DATA_BLOCK "IdentRfHmi"   // DB213
// stored: MemoryReserve 100
   VAR
      unitIdentRf : Array[0.."NO_OF_UNITS"] of "typeEMIdentRf";
   END_VAR
BEGIN
   unitIdentRf[0].identRfEM[0..7].selectedUnit := 0;
   unitIdentRf[0].identRfEM[0..7].selectedEM := 0;
   unitIdentRf[0].identRfEM[0..7].rfReaderId := 0;
   unitIdentRf[0].identRfEM[0..7].numberOfRf := 0;
   unitIdentRf[0].identRfEM[0].rfReader[0..1].deviceName := WSTRING#'';
   unitIdentRf[0].identRfEM[1].rfReader[0..1].deviceName := WSTRING#'';
   unitIdentRf[0].identRfEM[2].rfReader[0..1].deviceName := WSTRING#'';
   unitIdentRf[0].identRfEM[3].rfReader[0..1].deviceName := WSTRING#'';
   unitIdentRf[0].identRfEM[4].rfReader[0..1].deviceName := WSTRING#'';
   unitIdentRf[0].identRfEM[5].rfReader[0..1].deviceName := WSTRING#'';
   unitIdentRf[0].identRfEM[6].rfReader[0..1].deviceName := WSTRING#'';
   unitIdentRf[0].identRfEM[7].rfReader[0..1].deviceName := WSTRING#'';
   unitIdentRf[0].identRfEM[0].rfReader[0..1].deviceType := WSTRING#'';
   unitIdentRf[0].identRfEM[1].rfReader[0..1].deviceType := WSTRING#'';
   unitIdentRf[0].identRfEM[2].rfReader[0..1].deviceType := WSTRING#'';
   unitIdentRf[0].identRfEM[3].rfReader[0..1].deviceType := WSTRING#'';
   unitIdentRf[0].identRfEM[4].rfReader[0..1].deviceType := WSTRING#'';
   unitIdentRf[0].identRfEM[5].rfReader[0..1].deviceType := WSTRING#'';
   unitIdentRf[0].identRfEM[6].rfReader[0..1].deviceType := WSTRING#'';
   unitIdentRf[0].identRfEM[7].rfReader[0..1].deviceType := WSTRING#'';
   unitIdentRf[0].identRfEM[0].rfReader[0..1].deviceId := 0;
   unitIdentRf[0].identRfEM[1].rfReader[0..1].deviceId := 0;
   unitIdentRf[0].identRfEM[2].rfReader[0..1].deviceId := 0;
   unitIdentRf[0].identRfEM[3].rfReader[0..1].deviceId := 0;
   unitIdentRf[0].identRfEM[4].rfReader[0..1].deviceId := 0;
   unitIdentRf[0].identRfEM[5].rfReader[0..1].deviceId := 0;
   unitIdentRf[0].identRfEM[6].rfReader[0..1].deviceId := 0;
   unitIdentRf[0].identRfEM[7].rfReader[0..1].deviceId := 0;
   unitIdentRf[0].identRfEM[0].rfReader[0..1].tagType := WSTRING#'';
   unitIdentRf[0].identRfEM[1].rfReader[0..1].tagType := WSTRING#'';
   unitIdentRf[0].identRfEM[2].rfReader[0..1].tagType := WSTRING#'';
   unitIdentRf[0].identRfEM[3].rfReader[0..1].tagType := WSTRING#'';
   unitIdentRf[0].identRfEM[4].rfReader[0..1].tagType := WSTRING#'';
   unitIdentRf[0].identRfEM[5].rfReader[0..1].tagType := WSTRING#'';
   unitIdentRf[0].identRfEM[6].rfReader[0..1].tagType := WSTRING#'';
   unitIdentRf[0].identRfEM[7].rfReader[0..1].tagType := WSTRING#'';
   unitIdentRf[0].identRfEM[0].rfReader[0..1].cameraMode := WSTRING#'';
   unitIdentRf[0].identRfEM[1].rfReader[0..1].cameraMode := WSTRING#'';
   unitIdentRf[0].identRfEM[2].rfReader[0..1].cameraMode := WSTRING#'';
   unitIdentRf[0].identRfEM[3].rfReader[0..1].cameraMode := WSTRING#'';
   unitIdentRf[0].identRfEM[4].rfReader[0..1].cameraMode := WSTRING#'';
   unitIdentRf[0].identRfEM[5].rfReader[0..1].cameraMode := WSTRING#'';
   unitIdentRf[0].identRfEM[6].rfReader[0..1].cameraMode := WSTRING#'';
   unitIdentRf[0].identRfEM[7].rfReader[0..1].cameraMode := WSTRING#'';
   unitIdentRf[0].identRfEM[0].rfReader[0..1].resultState := WSTRING#'';
   unitIdentRf[0].identRfEM[1].rfReader[0..1].resultState := WSTRING#'';
   unitIdentRf[0].identRfEM[2].rfReader[0..1].resultState := WSTRING#'';
   unitIdentRf[0].identRfEM[3].rfReader[0..1].resultState := WSTRING#'';
   unitIdentRf[0].identRfEM[4].rfReader[0..1].resultState := WSTRING#'';
   unitIdentRf[0].identRfEM[5].rfReader[0..1].resultState := WSTRING#'';
   unitIdentRf[0].identRfEM[6].rfReader[0..1].resultState := WSTRING#'';
   unitIdentRf[0].identRfEM[7].rfReader[0..1].resultState := WSTRING#'';
   unitIdentRf[0].identRfEM[0].rfReader[0..1].progNo := 0;
   unitIdentRf[0].identRfEM[1].rfReader[0..1].progNo := 0;
   unitIdentRf[0].identRfEM[2].rfReader[0..1].progNo := 0;
   unitIdentRf[0].identRfEM[3].rfReader[0..1].progNo := 0;
   unitIdentRf[0].identRfEM[4].rfReader[0..1].progNo := 0;
   unitIdentRf[0].identRfEM[5].rfReader[0..1].progNo := 0;
   unitIdentRf[0].identRfEM[6].rfReader[0..1].progNo := 0;
   unitIdentRf[0].identRfEM[7].rfReader[0..1].progNo := 0;
   unitIdentRf[0].identRfEM[0].rfReader[0..1].progNumberWrite := 0;
   unitIdentRf[0].identRfEM[1].rfReader[0..1].progNumberWrite := 0;
   unitIdentRf[0].identRfEM[2].rfReader[0..1].progNumberWrite := 0;
   unitIdentRf[0].identRfEM[3].rfReader[0..1].progNumberWrite := 0;
   unitIdentRf[0].identRfEM[4].rfReader[0..1].progNumberWrite := 0;
   unitIdentRf[0].identRfEM[5].rfReader[0..1].progNumberWrite := 0;
   unitIdentRf[0].identRfEM[6].rfReader[0..1].progNumberWrite := 0;
   unitIdentRf[0].identRfEM[7].rfReader[0..1].progNumberWrite := 0;
   unitIdentRf[0].identRfEM[0].rfReader[0..1].pushbutton := 16#0000;
   unitIdentRf[0].identRfEM[1].rfReader[0..1].pushbutton := 16#0000;
   unitIdentRf[0].identRfEM[2].rfReader[0..1].pushbutton := 16#0000;
   unitIdentRf[0].identRfEM[3].rfReader[0..1].pushbutton := 16#0000;
   unitIdentRf[0].identRfEM[4].rfReader[0..1].pushbutton := 16#0000;
   unitIdentRf[0].identRfEM[5].rfReader[0..1].pushbutton := 16#0000;
   unitIdentRf[0].identRfEM[6].rfReader[0..1].pushbutton := 16#0000;
   unitIdentRf[0].identRfEM[7].rfReader[0..1].pushbutton := 16#0000;
   unitIdentRf[0].identRfEM[0].rfReader[0..1].enablePushbutton := 16#0000;
   unitIdentRf[0].identRfEM[1].rfReader[0..1].enablePushbutton := 16#0000;
   unitIdentRf[0].identRfEM[2].rfReader[0..1].enablePushbutton := 16#0000;
   unitIdentRf[0].identRfEM[3].rfReader[0..1].enablePushbutton := 16#0000;
   unitIdentRf[0].identRfEM[4].rfReader[0..1].enablePushbutton := 16#0000;
   unitIdentRf[0].identRfEM[5].rfReader[0..1].enablePushbutton := 16#0000;
   unitIdentRf[0].identRfEM[6].rfReader[0..1].enablePushbutton := 16#0000;
   unitIdentRf[0].identRfEM[7].rfReader[0..1].enablePushbutton := 16#0000;
   unitIdentRf[0].identRfEM[0].rfReader[0..1].status := 16#0000;
   unitIdentRf[0].identRfEM[1].rfReader[0..1].status := 16#0000;
   unitIdentRf[0].identRfEM[2].rfReader[0..1].status := 16#0000;
   unitIdentRf[0].identRfEM[3].rfReader[0..1].status := 16#0000;
   unitIdentRf[0].identRfEM[4].rfReader[0..1].status := 16#0000;
   unitIdentRf[0].identRfEM[5].rfReader[0..1].status := 16#0000;
   unitIdentRf[0].identRfEM[6].rfReader[0..1].status := 16#0000;
   unitIdentRf[0].identRfEM[7].rfReader[0..1].status := 16#0000;
   unitIdentRf[0].identRfEM[0].rfReader[0..1].alarmCategorie := 0;
   unitIdentRf[0].identRfEM[1].rfReader[0..1].alarmCategorie := 0;
   unitIdentRf[0].identRfEM[2].rfReader[0..1].alarmCategorie := 0;
   unitIdentRf[0].identRfEM[3].rfReader[0..1].alarmCategorie := 0;
   unitIdentRf[0].identRfEM[4].rfReader[0..1].alarmCategorie := 0;
   unitIdentRf[0].identRfEM[5].rfReader[0..1].alarmCategorie := 0;
   unitIdentRf[0].identRfEM[6].rfReader[0..1].alarmCategorie := 0;
   unitIdentRf[0].identRfEM[7].rfReader[0..1].alarmCategorie := 0;
   unitIdentRf[0].identRfEM[0].rfReader[0..1].alarmNo := 0;
   unitIdentRf[0].identRfEM[1].rfReader[0..1].alarmNo := 0;
   unitIdentRf[0].identRfEM[2].rfReader[0..1].alarmNo := 0;
   unitIdentRf[0].identRfEM[3].rfReader[0..1].alarmNo := 0;
   unitIdentRf[0].identRfEM[4].rfReader[0..1].alarmNo := 0;
   unitIdentRf[0].identRfEM[5].rfReader[0..1].alarmNo := 0;
   unitIdentRf[0].identRfEM[6].rfReader[0..1].alarmNo := 0;
   unitIdentRf[0].identRfEM[7].rfReader[0..1].alarmNo := 0;
   unitIdentRf[0].identRfEM[0].rfReader[0..1].alarmCode := 16#0000_0000;
   unitIdentRf[0].identRfEM[1].rfReader[0..1].alarmCode := 16#0000_0000;
   unitIdentRf[0].identRfEM[2].rfReader[0..1].alarmCode := 16#0000_0000;
   unitIdentRf[0].identRfEM[3].rfReader[0..1].alarmCode := 16#0000_0000;
   unitIdentRf[0].identRfEM[4].rfReader[0..1].alarmCode := 16#0000_0000;
   unitIdentRf[0].identRfEM[5].rfReader[0..1].alarmCode := 16#0000_0000;
   unitIdentRf[0].identRfEM[6].rfReader[0..1].alarmCode := 16#0000_0000;
   unitIdentRf[0].identRfEM[7].rfReader[0..1].alarmCode := 16#0000_0000;
   unitIdentRf[0].identRfEM[0].rfReader[0..1].resultColor := 0;
   unitIdentRf[0].identRfEM[1].rfReader[0..1].resultColor := 0;
   unitIdentRf[0].identRfEM[2].rfReader[0..1].resultColor := 0;
   unitIdentRf[0].identRfEM[3].rfReader[0..1].resultColor := 0;
   unitIdentRf[0].identRfEM[4].rfReader[0..1].resultColor := 0;
   unitIdentRf[0].identRfEM[5].rfReader[0..1].resultColor := 0;
   unitIdentRf[0].identRfEM[6].rfReader[0..1].resultColor := 0;
   unitIdentRf[0].identRfEM[7].rfReader[0..1].resultColor := 0;
   unitIdentRf[0].identRfEM[0].rfReader[0..1].statusColorCode := 0;
   unitIdentRf[0].identRfEM[1].rfReader[0..1].statusColorCode := 0;
   unitIdentRf[0].identRfEM[2].rfReader[0..1].statusColorCode := 0;
   unitIdentRf[0].identRfEM[3].rfReader[0..1].statusColorCode := 0;
   unitIdentRf[0].identRfEM[4].rfReader[0..1].statusColorCode := 0;
   unitIdentRf[0].identRfEM[5].rfReader[0..1].statusColorCode := 0;
   unitIdentRf[0].identRfEM[6].rfReader[0..1].statusColorCode := 0;
   unitIdentRf[0].identRfEM[7].rfReader[0..1].statusColorCode := 0;
   unitIdentRf[0].identRfEM[0].rfReader[0..1].datRead1 := '';
   unitIdentRf[0].identRfEM[1].rfReader[0..1].datRead1 := '';
   unitIdentRf[0].identRfEM[2].rfReader[0..1].datRead1 := '';
   unitIdentRf[0].identRfEM[3].rfReader[0..1].datRead1 := '';
   unitIdentRf[0].identRfEM[4].rfReader[0..1].datRead1 := '';
   unitIdentRf[0].identRfEM[5].rfReader[0..1].datRead1 := '';
   unitIdentRf[0].identRfEM[6].rfReader[0..1].datRead1 := '';
   unitIdentRf[0].identRfEM[7].rfReader[0..1].datRead1 := '';
   unitIdentRf[0].identRfEM[0].rfReader[0..1].datRead2 := '';
   unitIdentRf[0].identRfEM[1].rfReader[0..1].datRead2 := '';
   unitIdentRf[0].identRfEM[2].rfReader[0..1].datRead2 := '';
   unitIdentRf[0].identRfEM[3].rfReader[0..1].datRead2 := '';
   unitIdentRf[0].identRfEM[4].rfReader[0..1].datRead2 := '';
   unitIdentRf[0].identRfEM[5].rfReader[0..1].datRead2 := '';
   unitIdentRf[0].identRfEM[6].rfReader[0..1].datRead2 := '';
   unitIdentRf[0].identRfEM[7].rfReader[0..1].datRead2 := '';
   unitIdentRf[0].identRfEM[0].rfReader[0..1].datRead3 := '';
   unitIdentRf[0].identRfEM[1].rfReader[0..1].datRead3 := '';
   unitIdentRf[0].identRfEM[2].rfReader[0..1].datRead3 := '';
   unitIdentRf[0].identRfEM[3].rfReader[0..1].datRead3 := '';
   unitIdentRf[0].identRfEM[4].rfReader[0..1].datRead3 := '';
   unitIdentRf[0].identRfEM[5].rfReader[0..1].datRead3 := '';
   unitIdentRf[0].identRfEM[6].rfReader[0..1].datRead3 := '';
   unitIdentRf[0].identRfEM[7].rfReader[0..1].datRead3 := '';
   unitIdentRf[0].identRfEM[0].rfReader[0..1].datRead4 := '';
   unitIdentRf[0].identRfEM[1].rfReader[0..1].datRead4 := '';
   unitIdentRf[0].identRfEM[2].rfReader[0..1].datRead4 := '';
   unitIdentRf[0].identRfEM[3].rfReader[0..1].datRead4 := '';
   unitIdentRf[0].identRfEM[4].rfReader[0..1].datRead4 := '';
   unitIdentRf[0].identRfEM[5].rfReader[0..1].datRead4 := '';
   unitIdentRf[0].identRfEM[6].rfReader[0..1].datRead4 := '';
   unitIdentRf[0].identRfEM[7].rfReader[0..1].datRead4 := '';
   unitIdentRf[0].identRfEM[0].rfReader[0..1].datWrite1 := '';
   unitIdentRf[0].identRfEM[1].rfReader[0..1].datWrite1 := '';
   unitIdentRf[0].identRfEM[2].rfReader[0..1].datWrite1 := '';
   unitIdentRf[0].identRfEM[3].rfReader[0..1].datWrite1 := '';
   unitIdentRf[0].identRfEM[4].rfReader[0..1].datWrite1 := '';
   unitIdentRf[0].identRfEM[5].rfReader[0..1].datWrite1 := '';
   unitIdentRf[0].identRfEM[6].rfReader[0..1].datWrite1 := '';
   unitIdentRf[0].identRfEM[7].rfReader[0..1].datWrite1 := '';
   unitIdentRf[0].identRfEM[0].rfReader[0..1].datWrite2 := '';
   unitIdentRf[0].identRfEM[1].rfReader[0..1].datWrite2 := '';
   unitIdentRf[0].identRfEM[2].rfReader[0..1].datWrite2 := '';
   unitIdentRf[0].identRfEM[3].rfReader[0..1].datWrite2 := '';
   unitIdentRf[0].identRfEM[4].rfReader[0..1].datWrite2 := '';
   unitIdentRf[0].identRfEM[5].rfReader[0..1].datWrite2 := '';
   unitIdentRf[0].identRfEM[6].rfReader[0..1].datWrite2 := '';
   unitIdentRf[0].identRfEM[7].rfReader[0..1].datWrite2 := '';
   unitIdentRf[0].identRfEM[0].rfReader[0..1].datWrite3 := '';
   unitIdentRf[0].identRfEM[1].rfReader[0..1].datWrite3 := '';
   unitIdentRf[0].identRfEM[2].rfReader[0..1].datWrite3 := '';
   unitIdentRf[0].identRfEM[3].rfReader[0..1].datWrite3 := '';
   unitIdentRf[0].identRfEM[4].rfReader[0..1].datWrite3 := '';
   unitIdentRf[0].identRfEM[5].rfReader[0..1].datWrite3 := '';
   unitIdentRf[0].identRfEM[6].rfReader[0..1].datWrite3 := '';
   unitIdentRf[0].identRfEM[7].rfReader[0..1].datWrite3 := '';
   unitIdentRf[0].identRfEM[0].rfReader[0..1].datWrite4 := '';
   unitIdentRf[0].identRfEM[1].rfReader[0..1].datWrite4 := '';
   unitIdentRf[0].identRfEM[2].rfReader[0..1].datWrite4 := '';
   unitIdentRf[0].identRfEM[3].rfReader[0..1].datWrite4 := '';
   unitIdentRf[0].identRfEM[4].rfReader[0..1].datWrite4 := '';
   unitIdentRf[0].identRfEM[5].rfReader[0..1].datWrite4 := '';
   unitIdentRf[0].identRfEM[6].rfReader[0..1].datWrite4 := '';
   unitIdentRf[0].identRfEM[7].rfReader[0..1].datWrite4 := '';
END_DATA_BLOCK

DATA_BLOCK "IdentMvHmi"   // DB214
// stored: MemoryReserve 100
   VAR
      unitIdentMv : Array[0.."NO_OF_UNITS"] of "typeEMIdentMv";
   END_VAR
BEGIN
   unitIdentMv[0].identMvEM[0..7].selectedUnit := 0;
   unitIdentMv[0].identMvEM[0..7].selectedEM := 0;
   unitIdentMv[0].identMvEM[0..7].mvReaderId := 0;
   unitIdentMv[0].identMvEM[0..7].numberOfMv := 0;
   unitIdentMv[0].identMvEM[0].mvReader[0..1].deviceName := WSTRING#'';
   unitIdentMv[0].identMvEM[1].mvReader[0..1].deviceName := WSTRING#'';
   unitIdentMv[0].identMvEM[2].mvReader[0..1].deviceName := WSTRING#'';
   unitIdentMv[0].identMvEM[3].mvReader[0..1].deviceName := WSTRING#'';
   unitIdentMv[0].identMvEM[4].mvReader[0..1].deviceName := WSTRING#'';
   unitIdentMv[0].identMvEM[5].mvReader[0..1].deviceName := WSTRING#'';
   unitIdentMv[0].identMvEM[6].mvReader[0..1].deviceName := WSTRING#'';
   unitIdentMv[0].identMvEM[7].mvReader[0..1].deviceName := WSTRING#'';
   unitIdentMv[0].identMvEM[0].mvReader[0..1].deviceType := WSTRING#'';
   unitIdentMv[0].identMvEM[1].mvReader[0..1].deviceType := WSTRING#'';
   unitIdentMv[0].identMvEM[2].mvReader[0..1].deviceType := WSTRING#'';
   unitIdentMv[0].identMvEM[3].mvReader[0..1].deviceType := WSTRING#'';
   unitIdentMv[0].identMvEM[4].mvReader[0..1].deviceType := WSTRING#'';
   unitIdentMv[0].identMvEM[5].mvReader[0..1].deviceType := WSTRING#'';
   unitIdentMv[0].identMvEM[6].mvReader[0..1].deviceType := WSTRING#'';
   unitIdentMv[0].identMvEM[7].mvReader[0..1].deviceType := WSTRING#'';
   unitIdentMv[0].identMvEM[0].mvReader[0..1].deviceId := 0;
   unitIdentMv[0].identMvEM[1].mvReader[0..1].deviceId := 0;
   unitIdentMv[0].identMvEM[2].mvReader[0..1].deviceId := 0;
   unitIdentMv[0].identMvEM[3].mvReader[0..1].deviceId := 0;
   unitIdentMv[0].identMvEM[4].mvReader[0..1].deviceId := 0;
   unitIdentMv[0].identMvEM[5].mvReader[0..1].deviceId := 0;
   unitIdentMv[0].identMvEM[6].mvReader[0..1].deviceId := 0;
   unitIdentMv[0].identMvEM[7].mvReader[0..1].deviceId := 0;
   unitIdentMv[0].identMvEM[0].mvReader[0..1].tagType := WSTRING#'';
   unitIdentMv[0].identMvEM[1].mvReader[0..1].tagType := WSTRING#'';
   unitIdentMv[0].identMvEM[2].mvReader[0..1].tagType := WSTRING#'';
   unitIdentMv[0].identMvEM[3].mvReader[0..1].tagType := WSTRING#'';
   unitIdentMv[0].identMvEM[4].mvReader[0..1].tagType := WSTRING#'';
   unitIdentMv[0].identMvEM[5].mvReader[0..1].tagType := WSTRING#'';
   unitIdentMv[0].identMvEM[6].mvReader[0..1].tagType := WSTRING#'';
   unitIdentMv[0].identMvEM[7].mvReader[0..1].tagType := WSTRING#'';
   unitIdentMv[0].identMvEM[0].mvReader[0..1].cameraMode := WSTRING#'';
   unitIdentMv[0].identMvEM[1].mvReader[0..1].cameraMode := WSTRING#'';
   unitIdentMv[0].identMvEM[2].mvReader[0..1].cameraMode := WSTRING#'';
   unitIdentMv[0].identMvEM[3].mvReader[0..1].cameraMode := WSTRING#'';
   unitIdentMv[0].identMvEM[4].mvReader[0..1].cameraMode := WSTRING#'';
   unitIdentMv[0].identMvEM[5].mvReader[0..1].cameraMode := WSTRING#'';
   unitIdentMv[0].identMvEM[6].mvReader[0..1].cameraMode := WSTRING#'';
   unitIdentMv[0].identMvEM[7].mvReader[0..1].cameraMode := WSTRING#'';
   unitIdentMv[0].identMvEM[0].mvReader[0..1].resultState := WSTRING#'';
   unitIdentMv[0].identMvEM[1].mvReader[0..1].resultState := WSTRING#'';
   unitIdentMv[0].identMvEM[2].mvReader[0..1].resultState := WSTRING#'';
   unitIdentMv[0].identMvEM[3].mvReader[0..1].resultState := WSTRING#'';
   unitIdentMv[0].identMvEM[4].mvReader[0..1].resultState := WSTRING#'';
   unitIdentMv[0].identMvEM[5].mvReader[0..1].resultState := WSTRING#'';
   unitIdentMv[0].identMvEM[6].mvReader[0..1].resultState := WSTRING#'';
   unitIdentMv[0].identMvEM[7].mvReader[0..1].resultState := WSTRING#'';
   unitIdentMv[0].identMvEM[0].mvReader[0..1].progNo := 0;
   unitIdentMv[0].identMvEM[1].mvReader[0..1].progNo := 0;
   unitIdentMv[0].identMvEM[2].mvReader[0..1].progNo := 0;
   unitIdentMv[0].identMvEM[3].mvReader[0..1].progNo := 0;
   unitIdentMv[0].identMvEM[4].mvReader[0..1].progNo := 0;
   unitIdentMv[0].identMvEM[5].mvReader[0..1].progNo := 0;
   unitIdentMv[0].identMvEM[6].mvReader[0..1].progNo := 0;
   unitIdentMv[0].identMvEM[7].mvReader[0..1].progNo := 0;
   unitIdentMv[0].identMvEM[0].mvReader[0..1].progNumberWrite := 0;
   unitIdentMv[0].identMvEM[1].mvReader[0..1].progNumberWrite := 0;
   unitIdentMv[0].identMvEM[2].mvReader[0..1].progNumberWrite := 0;
   unitIdentMv[0].identMvEM[3].mvReader[0..1].progNumberWrite := 0;
   unitIdentMv[0].identMvEM[4].mvReader[0..1].progNumberWrite := 0;
   unitIdentMv[0].identMvEM[5].mvReader[0..1].progNumberWrite := 0;
   unitIdentMv[0].identMvEM[6].mvReader[0..1].progNumberWrite := 0;
   unitIdentMv[0].identMvEM[7].mvReader[0..1].progNumberWrite := 0;
   unitIdentMv[0].identMvEM[0].mvReader[0..1].pushbutton := 16#0000;
   unitIdentMv[0].identMvEM[1].mvReader[0..1].pushbutton := 16#0000;
   unitIdentMv[0].identMvEM[2].mvReader[0..1].pushbutton := 16#0000;
   unitIdentMv[0].identMvEM[3].mvReader[0..1].pushbutton := 16#0000;
   unitIdentMv[0].identMvEM[4].mvReader[0..1].pushbutton := 16#0000;
   unitIdentMv[0].identMvEM[5].mvReader[0..1].pushbutton := 16#0000;
   unitIdentMv[0].identMvEM[6].mvReader[0..1].pushbutton := 16#0000;
   unitIdentMv[0].identMvEM[7].mvReader[0..1].pushbutton := 16#0000;
   unitIdentMv[0].identMvEM[0].mvReader[0..1].enablePushbutton := 16#0000;
   unitIdentMv[0].identMvEM[1].mvReader[0..1].enablePushbutton := 16#0000;
   unitIdentMv[0].identMvEM[2].mvReader[0..1].enablePushbutton := 16#0000;
   unitIdentMv[0].identMvEM[3].mvReader[0..1].enablePushbutton := 16#0000;
   unitIdentMv[0].identMvEM[4].mvReader[0..1].enablePushbutton := 16#0000;
   unitIdentMv[0].identMvEM[5].mvReader[0..1].enablePushbutton := 16#0000;
   unitIdentMv[0].identMvEM[6].mvReader[0..1].enablePushbutton := 16#0000;
   unitIdentMv[0].identMvEM[7].mvReader[0..1].enablePushbutton := 16#0000;
   unitIdentMv[0].identMvEM[0].mvReader[0..1].status := 16#0000;
   unitIdentMv[0].identMvEM[1].mvReader[0..1].status := 16#0000;
   unitIdentMv[0].identMvEM[2].mvReader[0..1].status := 16#0000;
   unitIdentMv[0].identMvEM[3].mvReader[0..1].status := 16#0000;
   unitIdentMv[0].identMvEM[4].mvReader[0..1].status := 16#0000;
   unitIdentMv[0].identMvEM[5].mvReader[0..1].status := 16#0000;
   unitIdentMv[0].identMvEM[6].mvReader[0..1].status := 16#0000;
   unitIdentMv[0].identMvEM[7].mvReader[0..1].status := 16#0000;
   unitIdentMv[0].identMvEM[0].mvReader[0..1].alarmCategorie := 0;
   unitIdentMv[0].identMvEM[1].mvReader[0..1].alarmCategorie := 0;
   unitIdentMv[0].identMvEM[2].mvReader[0..1].alarmCategorie := 0;
   unitIdentMv[0].identMvEM[3].mvReader[0..1].alarmCategorie := 0;
   unitIdentMv[0].identMvEM[4].mvReader[0..1].alarmCategorie := 0;
   unitIdentMv[0].identMvEM[5].mvReader[0..1].alarmCategorie := 0;
   unitIdentMv[0].identMvEM[6].mvReader[0..1].alarmCategorie := 0;
   unitIdentMv[0].identMvEM[7].mvReader[0..1].alarmCategorie := 0;
   unitIdentMv[0].identMvEM[0].mvReader[0..1].alarmNo := 0;
   unitIdentMv[0].identMvEM[1].mvReader[0..1].alarmNo := 0;
   unitIdentMv[0].identMvEM[2].mvReader[0..1].alarmNo := 0;
   unitIdentMv[0].identMvEM[3].mvReader[0..1].alarmNo := 0;
   unitIdentMv[0].identMvEM[4].mvReader[0..1].alarmNo := 0;
   unitIdentMv[0].identMvEM[5].mvReader[0..1].alarmNo := 0;
   unitIdentMv[0].identMvEM[6].mvReader[0..1].alarmNo := 0;
   unitIdentMv[0].identMvEM[7].mvReader[0..1].alarmNo := 0;
   unitIdentMv[0].identMvEM[0].mvReader[0..1].alarmCode := 16#0000_0000;
   unitIdentMv[0].identMvEM[1].mvReader[0..1].alarmCode := 16#0000_0000;
   unitIdentMv[0].identMvEM[2].mvReader[0..1].alarmCode := 16#0000_0000;
   unitIdentMv[0].identMvEM[3].mvReader[0..1].alarmCode := 16#0000_0000;
   unitIdentMv[0].identMvEM[4].mvReader[0..1].alarmCode := 16#0000_0000;
   unitIdentMv[0].identMvEM[5].mvReader[0..1].alarmCode := 16#0000_0000;
   unitIdentMv[0].identMvEM[6].mvReader[0..1].alarmCode := 16#0000_0000;
   unitIdentMv[0].identMvEM[7].mvReader[0..1].alarmCode := 16#0000_0000;
   unitIdentMv[0].identMvEM[0].mvReader[0..1].resultColor := 0;
   unitIdentMv[0].identMvEM[1].mvReader[0..1].resultColor := 0;
   unitIdentMv[0].identMvEM[2].mvReader[0..1].resultColor := 0;
   unitIdentMv[0].identMvEM[3].mvReader[0..1].resultColor := 0;
   unitIdentMv[0].identMvEM[4].mvReader[0..1].resultColor := 0;
   unitIdentMv[0].identMvEM[5].mvReader[0..1].resultColor := 0;
   unitIdentMv[0].identMvEM[6].mvReader[0..1].resultColor := 0;
   unitIdentMv[0].identMvEM[7].mvReader[0..1].resultColor := 0;
   unitIdentMv[0].identMvEM[0].mvReader[0..1].statusColorCode := 0;
   unitIdentMv[0].identMvEM[1].mvReader[0..1].statusColorCode := 0;
   unitIdentMv[0].identMvEM[2].mvReader[0..1].statusColorCode := 0;
   unitIdentMv[0].identMvEM[3].mvReader[0..1].statusColorCode := 0;
   unitIdentMv[0].identMvEM[4].mvReader[0..1].statusColorCode := 0;
   unitIdentMv[0].identMvEM[5].mvReader[0..1].statusColorCode := 0;
   unitIdentMv[0].identMvEM[6].mvReader[0..1].statusColorCode := 0;
   unitIdentMv[0].identMvEM[7].mvReader[0..1].statusColorCode := 0;
   unitIdentMv[0].identMvEM[0].mvReader[0..1].datRead1 := '';
   unitIdentMv[0].identMvEM[1].mvReader[0..1].datRead1 := '';
   unitIdentMv[0].identMvEM[2].mvReader[0..1].datRead1 := '';
   unitIdentMv[0].identMvEM[3].mvReader[0..1].datRead1 := '';
   unitIdentMv[0].identMvEM[4].mvReader[0..1].datRead1 := '';
   unitIdentMv[0].identMvEM[5].mvReader[0..1].datRead1 := '';
   unitIdentMv[0].identMvEM[6].mvReader[0..1].datRead1 := '';
   unitIdentMv[0].identMvEM[7].mvReader[0..1].datRead1 := '';
   unitIdentMv[0].identMvEM[0].mvReader[0..1].datRead2 := '';
   unitIdentMv[0].identMvEM[1].mvReader[0..1].datRead2 := '';
   unitIdentMv[0].identMvEM[2].mvReader[0..1].datRead2 := '';
   unitIdentMv[0].identMvEM[3].mvReader[0..1].datRead2 := '';
   unitIdentMv[0].identMvEM[4].mvReader[0..1].datRead2 := '';
   unitIdentMv[0].identMvEM[5].mvReader[0..1].datRead2 := '';
   unitIdentMv[0].identMvEM[6].mvReader[0..1].datRead2 := '';
   unitIdentMv[0].identMvEM[7].mvReader[0..1].datRead2 := '';
   unitIdentMv[0].identMvEM[0].mvReader[0..1].datRead3 := '';
   unitIdentMv[0].identMvEM[1].mvReader[0..1].datRead3 := '';
   unitIdentMv[0].identMvEM[2].mvReader[0..1].datRead3 := '';
   unitIdentMv[0].identMvEM[3].mvReader[0..1].datRead3 := '';
   unitIdentMv[0].identMvEM[4].mvReader[0..1].datRead3 := '';
   unitIdentMv[0].identMvEM[5].mvReader[0..1].datRead3 := '';
   unitIdentMv[0].identMvEM[6].mvReader[0..1].datRead3 := '';
   unitIdentMv[0].identMvEM[7].mvReader[0..1].datRead3 := '';
   unitIdentMv[0].identMvEM[0].mvReader[0..1].datRead4 := '';
   unitIdentMv[0].identMvEM[1].mvReader[0..1].datRead4 := '';
   unitIdentMv[0].identMvEM[2].mvReader[0..1].datRead4 := '';
   unitIdentMv[0].identMvEM[3].mvReader[0..1].datRead4 := '';
   unitIdentMv[0].identMvEM[4].mvReader[0..1].datRead4 := '';
   unitIdentMv[0].identMvEM[5].mvReader[0..1].datRead4 := '';
   unitIdentMv[0].identMvEM[6].mvReader[0..1].datRead4 := '';
   unitIdentMv[0].identMvEM[7].mvReader[0..1].datRead4 := '';
   unitIdentMv[0].identMvEM[0].mvReader[0].datWrite1 := '';
   unitIdentMv[0].identMvEM[0].mvReader[1].datWrite1 := 'Siemens';
   unitIdentMv[0].identMvEM[1].mvReader[0..1].datWrite1 := '';
   unitIdentMv[0].identMvEM[2].mvReader[0..1].datWrite1 := '';
   unitIdentMv[0].identMvEM[3].mvReader[0..1].datWrite1 := '';
   unitIdentMv[0].identMvEM[4].mvReader[0..1].datWrite1 := '';
   unitIdentMv[0].identMvEM[5].mvReader[0..1].datWrite1 := '';
   unitIdentMv[0].identMvEM[6].mvReader[0..1].datWrite1 := '';
   unitIdentMv[0].identMvEM[7].mvReader[0..1].datWrite1 := '';
   unitIdentMv[0].identMvEM[0].mvReader[0..1].datWrite2 := '';
   unitIdentMv[0].identMvEM[1].mvReader[0..1].datWrite2 := '';
   unitIdentMv[0].identMvEM[2].mvReader[0..1].datWrite2 := '';
   unitIdentMv[0].identMvEM[3].mvReader[0..1].datWrite2 := '';
   unitIdentMv[0].identMvEM[4].mvReader[0..1].datWrite2 := '';
   unitIdentMv[0].identMvEM[5].mvReader[0..1].datWrite2 := '';
   unitIdentMv[0].identMvEM[6].mvReader[0..1].datWrite2 := '';
   unitIdentMv[0].identMvEM[7].mvReader[0..1].datWrite2 := '';
   unitIdentMv[0].identMvEM[0].mvReader[0..1].datWrite3 := '';
   unitIdentMv[0].identMvEM[1].mvReader[0..1].datWrite3 := '';
   unitIdentMv[0].identMvEM[2].mvReader[0..1].datWrite3 := '';
   unitIdentMv[0].identMvEM[3].mvReader[0..1].datWrite3 := '';
   unitIdentMv[0].identMvEM[4].mvReader[0..1].datWrite3 := '';
   unitIdentMv[0].identMvEM[5].mvReader[0..1].datWrite3 := '';
   unitIdentMv[0].identMvEM[6].mvReader[0..1].datWrite3 := '';
   unitIdentMv[0].identMvEM[7].mvReader[0..1].datWrite3 := '';
   unitIdentMv[0].identMvEM[0].mvReader[0..1].datWrite4 := '';
   unitIdentMv[0].identMvEM[1].mvReader[0..1].datWrite4 := '';
   unitIdentMv[0].identMvEM[2].mvReader[0..1].datWrite4 := '';
   unitIdentMv[0].identMvEM[3].mvReader[0..1].datWrite4 := '';
   unitIdentMv[0].identMvEM[4].mvReader[0..1].datWrite4 := '';
   unitIdentMv[0].identMvEM[5].mvReader[0..1].datWrite4 := '';
   unitIdentMv[0].identMvEM[6].mvReader[0..1].datWrite4 := '';
   unitIdentMv[0].identMvEM[7].mvReader[0..1].datWrite4 := '';
END_DATA_BLOCK

DATA_BLOCK "BK02"   // DB304
// stored: MemoryReserve 100
   VAR
      "X10-1.SUCTION PAD TOP DOWN" : Bool := TRUE;
      "X11-1.SUCTION PAD BTM DOWN" : Bool := TRUE;
      "X12-1.CUTTER DOWN" : Bool := TRUE;
      "X13-1.TAPE TOP DOWN" : Bool := FALSE;
      "X14-1.TAPE BTM DOWN" : Bool := TRUE;
      "X15-1.SPLICE HEAD ROTATE TOP BACKWARD" : Bool := TRUE;
      "X16-1.SPLICE HEAD ROTATE BTM BACKWARD" : Bool := TRUE;
      "X17-1.SPARE" : Bool := FALSE;
      "X10-2.SUCTION PAD TOP UP" : Bool := FALSE;
      "X11-2.SUCTION PAD BTM UP" : Bool := FALSE;
      "X12-2.CUTTER UP" : Bool := FALSE;
      "X13-2.TAPE TOP UP" : Bool := TRUE;
      "X14-2.TAPE BTM UP" : Bool := FALSE;
      "X15-2.SPLICE HEAD ROTATE TOP FORWARD" : Bool := FALSE;
      "X16-2.SPLICE HEAD ROTATE BTM FORWARD" : Bool := FALSE;
      "X17-2.SPARE" : Bool := FALSE;
   END_VAR
BEGIN
END_DATA_BLOCK

DATA_BLOCK "BK04"   // DB308
// stored: MemoryReserve 100
   VAR
      "X10-1.CATHODE MAIN P&P1 LIMITS SENSOR(-)" : Bool := TRUE;
      "X11-1.CATHODE MAIN P&P1 LIMITS SENSOR(+)" : Bool := TRUE;
      "X12-1.CATHODE MAIN P&P2 LIMITS SENSOR(-)" : Bool := TRUE;
      "X13-1.CATHODE MAIN P&P2 LIMITS SENSOR(+)" : Bool := TRUE;
      "X14-1.ANODE MAIN P&P2 LIMITS SENSOR(-)" : Bool := TRUE;
      "X15-1.ANODE MAIN P&P2 LIMITS SENSOR(+)" : Bool := TRUE;
      "X16-1.ANODE MAIN P&P1 LIMITS SENSOR(-)" : Bool := TRUE;
      "X17-1.ANODE MAIN P&P1 LIMITS SENSOR(+)" : Bool := TRUE;
      "X10-2.CATHODE MAIN P&P1 LIMITS SENSOR HOME" : Bool := TRUE;
      "X11-2.SPARE" : Bool := FALSE;
      "X12-2.CATHODE MAIN P&P2 LIMITS SENSOR HOME" : Bool := TRUE;
      "X13-2.SPARE" : Bool := FALSE;
      "X14-2.ANODE MAIN P&P2 LIMITS SENSOR HOME" : Bool := TRUE;
      "X15-2.SPARE" : Bool := FALSE;
      "X16-2.ANODE MAIN P&P1 LIMITS SENSOR HOME" : Bool := TRUE;
      "X17-2.SPARE" : Bool := FALSE;
   END_VAR
BEGIN
END_DATA_BLOCK

DATA_BLOCK "BK10"   // DB306
// stored: MemoryReserve 100
   VAR
      "X10-1.ANODE FIX FRONT BACKWARD" : Bool := TRUE;
      "X11-1.SEPA CLAMP SAFETY PIN DETECT SENSOR" : Bool := FALSE;
      "X12-1.ANODE FIX REAR BACKWARD" : Bool := TRUE;
      "X13-1.SEPA CLAMP PRESSURE SWITCH" : Bool := FALSE;
      "X14-1.FIX ANODE DETECT SENSOR" : Bool := FALSE;
      "X15-1.SPARE" : Bool := FALSE;
      "X16-1.SPARE" : Bool := FALSE;
      "X17-1.SPARE" : Bool := FALSE;
      "X10-2.ANODE FIX FRONT FORWARD" : Bool := FALSE;
      "X11-2.SEPA GRIPPER SAFETY PIN DETECT SENSOR" : Bool := FALSE;
      "X12-2.ANODE FIX REAR FORWARD" : Bool := FALSE;
      "X13-2.SPARE" : Bool := FALSE;
      "X14-2.SPARE" : Bool := FALSE;
      "X15-2.SPARE" : Bool := FALSE;
      "X16-2.SPARE" : Bool := FALSE;
      "X17-2.SPARE" : Bool := FALSE;
   END_VAR
BEGIN
END_DATA_BLOCK

DATA_BLOCK "BK11"   // DB305
// stored: MemoryReserve 100
   VAR
      "X10-1.ANODE NG BOX FULL SENSOR" : Bool := TRUE;
      "X10-2.SPARE" : Bool := FALSE;
      "X12-1.ANODE NG BOX LIFT DOWN" : Bool := FALSE;
      "X12-2.ANODE NG BOX LIFT UP" : Bool := TRUE;
      "X14-1.ANODE NG BOX LOCK DOWN" : Bool := TRUE;
      "X14-2.ANODE NG BOX LOCK UP" : Bool := FALSE;
      "X16-1.ANODE NG BOX NG BOX DETECT SENSOR" : Bool := TRUE;
      "X16-2.SPARE" : Bool := FALSE;
   END_VAR
BEGIN
END_DATA_BLOCK

DATA_BLOCK "BK13"   // DB282
// stored: MemoryReserve 100
   VAR
      "X10-1.CATHODE ALIGN TABLE Y1-AXIS LIMIT SENSOR(-)" : Bool := TRUE;
      "X11-1.CATHODE ALIGN TABLE Y1-AXIS LIMIT SENSOR(+)" : Bool := TRUE;
      "X12-1.CATHODE ALIGN TABLE X-AXIS LIMIT SENSOR(-)" : Bool := TRUE;
      "X13-1.CATHODE ALIGN TABLE X-AXIS LIMIT SENSOR(+)" : Bool := TRUE;
      "X14-1.CATHODE ALIGN TABLE Y2-AXIS LIMIT SENSOR(-)" : Bool := TRUE;
      "X15-1.CATHODE ALIGN TABLE Y2-AXIS LIMIT SENSOR(+)" : Bool := TRUE;
      "X16-1.CATHODE ALIGN TABLE ELECTRODE DETECT SENSOR" : Bool := FALSE;
      "X17-1.CATHODE ALIGN TABLE PRESSURE SWITCH" : Bool := FALSE;
      "X10-2.CATHODE ALIGN TABLE Y1-AXIS HOME SENSOR" : Bool := TRUE;
      "X11-2.SPARE" : Bool := FALSE;
      "X12-2.CATHODE ALIGN TABLE X-AXIS HOME SENSOR" : Bool := FALSE;
      "X13-2.SPARE" : Bool := FALSE;
      "X14-2.CATHODE ALIGN TABLE Y2-AXIS HOME SENSOR" : Bool := FALSE;
      "X15-2.SPARE" : Bool := FALSE;
      "X16-2.SPARE" : Bool := FALSE;
      "X17-2.SPARE" : Bool := FALSE;
   END_VAR
BEGIN
END_DATA_BLOCK

DATA_BLOCK "BK18"   // DB312
// stored: MemoryReserve 100
   VAR
      "X10-1.ANODE MANDREL REAR Y AXIS LIMIT SENSOR(-)" : Bool := TRUE;
      "X11-1.ANODE MANDREL REAR Y AXIS LIMIT SENSOR(+)" : Bool := TRUE;
      "X12-1.ANODE MANDREL REAR Z AXIS LIMIT SENSOR(-)" : Bool := TRUE;
      "X13-1.ANODE MANDREL REAR Z AXIS LIMIT SENSOR(+)" : Bool := TRUE;
      "X14-1.ANODE MANDREL FRONT Y AXIS LIMIT SENSOR(-)" : Bool := TRUE;
      "X15-1.ANODE MANDREL FRONT Y AXIS LIMIT SENSOR(+)" : Bool := TRUE;
      "X16-1.ANODE MANDREL FRONT Z AXIS LIMIT SENSOR(-)" : Bool := TRUE;
      "X17-1.ANODE MANDREL FRONT Z AXIS LIMIT SENSOR(+)" : Bool := TRUE;
      "X10-2.ANODE MANDREL REAR Y AXIS HOME SENSOR" : Bool := TRUE;
      "X11-2.SPARE" : Bool := FALSE;
      "X12-2.ANODE MANDREL REAR Z AXIS HOME SENSOR" : Bool := TRUE;
      "X13-2.SPARE" : Bool := FALSE;
      "X14-2.ANODE MANDREL FRONT Y AXIS HOME SENSOR" : Bool := TRUE;
      "X15-2.SPARE" : Bool := FALSE;
      "X16-2.ANODE MANDREL FRONT Z AXIS HOME SENSOR" : Bool := TRUE;
      "X17-2.SPARE" : Bool := FALSE;
   END_VAR
BEGIN
END_DATA_BLOCK

DATA_BLOCK "BK20"   // DB311
// stored: MemoryReserve 100
   VAR
      "X10-1.STACK TABLE Z-AXIS LIMIT SENSOR(-)" : Bool := TRUE;
      "X11-1.STACK TABLE Z-AXIS LIMIT SENSOR(+)" : Bool := TRUE;
      "X12-1.STACK TABLE GAP PAD DOWN" : Bool := TRUE;
      "X13-1.STACK TABLE GAP PAD UP" : Bool := FALSE;
      "X14-1.STACK TABLE OUT FRONT Z-AXIS LIMIT SENSOR(-)" : Bool := TRUE;
      "X15-1.STACK TABLE OUT FRONT Z-AXIS LIMIT SENSOR(+)" : Bool := TRUE;
      "X16-1.STACK TABLE VACUUM PRESSURE SWITCH" : Bool := FALSE;
      "X17-1.SPARE" : Bool := FALSE;
      "X10-2.STACK TABLE Z-AXIS HOME SENSOR" : Bool := TRUE;
      "X11-2.SPARE" : Bool := FALSE;
      "X12-2.SPARE" : Bool := FALSE;
      "X13-2.SPARE" : Bool := FALSE;
      "X14-2.STACK TABLE OUT FRONT Z-AXIS HOME SENSOR" : Bool := TRUE;
      "X15-2.SPARE" : Bool := FALSE;
      "X16-2.STACK TABLE ELECTRODE DETECT SENSOR" : Bool := FALSE;
      "X17-2.SPARE" : Bool := FALSE;
   END_VAR
BEGIN
END_DATA_BLOCK

DATA_BLOCK "BK21"   // DB249
// stored: MemoryReserve 100
   VAR
      "X10-1.SEPA CLAMP&CUTTER X-AXIS LIMIT SENSOR(-)" : Bool := TRUE;
      "X10-2.SEPA CLAMP&CUTTER X-AXIS HOME SENSOR" : Bool := TRUE;
      "X12-1.SEPA CLAMP&CUTTER X-AXIS LIMIT SENSOR(+)" : Bool := TRUE;
      "X12-2.SPARE" : Bool := FALSE;
      "X14-1.SEPA GRIPPER X-AXIS LIMIT SENSOR(-)" : Bool := TRUE;
      "X14-2.SEPA GRIPPER X-AXIS HOME SENSOR" : Bool := TRUE;
      "X16-1.SEPA GRIPPER X-AXIS LIMIT SENSOR(+)" : Bool := TRUE;
      "X16-2.SPARE" : Bool := FALSE;
   END_VAR
BEGIN
END_DATA_BLOCK

DATA_BLOCK "BK22"   // DB274
// stored: MemoryReserve 100
   VAR
      "X10-1.SEPA GRIPPER CLAMP OPEN" : Bool := TRUE;
      "X11-1.SPARE" : Bool := FALSE;
      "X12-1.SEPA GRIPPER CLAMP DETECT SENSOR" : Bool := TRUE;
      "X13-1.SEPA GRIPPER BACKWARD" : Bool := FALSE;
      "X14-1.SEPA GRIPPER C-AXIS LIMIT SENSOR(-)" : Bool := TRUE;
      "X15-1.SEPA GRIPPER C-AXIS LIMIT SENSOR(+)" : Bool := TRUE;
      "X16-1.SEPA GRIPPER Z-AXIS LIMIT SENSOR(-)" : Bool := TRUE;
      "X17-1.SEPA GRIPPER Z-AXIS LIMIT SENSOR(+)" : Bool := TRUE;
      "X10-2.SEPA GRIPPER CLAMP CLOSE" : Bool := FALSE;
      "X11-2.SPARE" : Bool := FALSE;
      "X12-2.SPARE" : Bool := FALSE;
      "X13-2.SEPA GRIPPER FORWARD" : Bool := FALSE;
      "X14-2.SEPA GRIPPER C-AXIS HOME SENSOR" : Bool := TRUE;
      "X15-2.SPARE" : Bool := FALSE;
      "X16-2.SEPA GRIPPER Z-AXIS HOME SENSOR" : Bool := TRUE;
      "X17-2.SPARE" : Bool := FALSE;
   END_VAR
BEGIN
END_DATA_BLOCK

DATA_BLOCK "BK26"   // DB260
// stored: MemoryReserve 100
   VAR
      "X10-1.JR WINDER B-AXIS HOME SENSOR" : Bool := TRUE;
      "X11-1.JR WINDER CLAMP REAR TOP DOWN" : Bool := FALSE;
      "X12-1.MAIN VALVE DIGITAL PRESSURE SWITCH OUT1" : Bool := FALSE;
      "X13-1.JR WINDER CLAMP REAR BTM DOWN" : Bool := FALSE;
      "X14-1.SPARE" : Bool := FALSE;
      "X15-1.JR WINDER CLAMP TOP REAR PRESSURE SWITCH" : Bool := FALSE;
      "X16-1.SPARE" : Bool := FALSE;
      "X17-1.SPARE" : Bool := FALSE;
      "X10-2.SPARE" : Bool := FALSE;
      "X11-2.SPARE" : Bool := FALSE;
      "X12-2.MAIN VALVE DIGITAL PRESSURE SWITCH OUT2" : Bool := FALSE;
      "X13-2.SPARE" : Bool := FALSE;
      "X14-2.SPARE" : Bool := FALSE;
      "X15-2.JR WINDER CLAMP TOP FRONT PRESSURE SWITCH" : Bool := FALSE;
      "X16-2.SPARE" : Bool := FALSE;
      "X17-2.SPARE" : Bool := FALSE;
   END_VAR
BEGIN
END_DATA_BLOCK

DATA_BLOCK "BK27"   // DB255
// stored: MemoryReserve 100
   VAR
      "X10-1.SPARE" : Bool := FALSE;
      "X11-1.JR WINDER CLAMP FRONT TOP DOWN" : Bool := FALSE;
      "X12-1.SPARE" : Bool := FALSE;
      "X13-1.JR WINDER CLAMP FRONT BTM DOWN" : Bool := FALSE;
      "X14-1.SPARE" : Bool := FALSE;
      "X15-1.JR WINDER CLAMP FRONT TOP PRESSURE SWITCH" : Bool := FALSE;
      "X16-1.JR WINDER STACK DETECT SENSOR" : Bool := FALSE;
      "X17-1.SPARE" : Bool := FALSE;
      "X10-2.SPARE" : Bool := FALSE;
      "X11-2.SPARE" : Bool := FALSE;
      "X12-2.SPARE" : Bool := FALSE;
      "X13-2.SPARE" : Bool := FALSE;
      "X14-2.SPARE" : Bool := FALSE;
      "X15-2.JR WINDER CLAMP FRONT BTM PRESSURE SWITCH" : Bool := FALSE;
      "X16-2.SPARE" : Bool := FALSE;
      "X17-2.SPARE" : Bool := FALSE;
   END_VAR
BEGIN
END_DATA_BLOCK

DATA_BLOCK "BK31"   // DB279
// stored: MemoryReserve 100
   VAR
      "ANODE MAIN P&P1 VACUUM ON" : Bool := FALSE;
      "ANODE MAIN P&P1 VACUUM OFF" : Bool := FALSE;
      "ANODE MAIN P&P2 VACUUM ON" : Bool := FALSE;
      "ANODE MAIN P&P2 VACUUM OFF" : Bool := FALSE;
      "ANODE MAIN NG P&P VACUUM ON" : Bool := FALSE;
      "ANODE MAIN NG P&P VACUUM OFF" : Bool := FALSE;
      "ANODE ALIGN TABLE VACUUM ON" : Bool := FALSE;
      "ANODE ALIGN TABLE VACUUM OFF" : Bool := FALSE;
   END_VAR
BEGIN
END_DATA_BLOCK

DATA_BLOCK "BK33"   // DB236
// stored: MemoryReserve 100
   VAR
      SPARE : Bool := FALSE;
      SPARE_1 : Bool := FALSE;
      SPARE_2 : Bool := FALSE;
      SPARE_3 : Bool := FALSE;
      SPARE_4 : Bool := FALSE;
      SPARE_5 : Bool := FALSE;
      SPARE_6 : Bool := FALSE;
      SPARE_7 : Bool := FALSE;
   END_VAR
BEGIN
END_DATA_BLOCK

ORGANIZATION_BLOCK "Main"   // OB1, LAD, ProgramCycle
TITLE = "Main Program Sweep (Cycle)"
// stored: AutoNumber false, IsIECCheckEnabled true, SetENOAutomatically true
   VAR_INPUT
      Initial_Call : Bool;   // Initial call of this OB
      Remanence : Bool;   // =True, if remanent data are available
   END_VAR
   VAR_TEMP   // added for the SCL form of the ladder/FBD networks
      _w1 : Bool;
      _w2 : Bool;
      _w3 : Bool;
      _w4 : Bool;
      _w5 : Bool;
      _w6 : Bool;
   END_VAR
BEGIN

REGION Network 1: First Cycle
   // Set bit to true in first cycle, and false in all other cycles
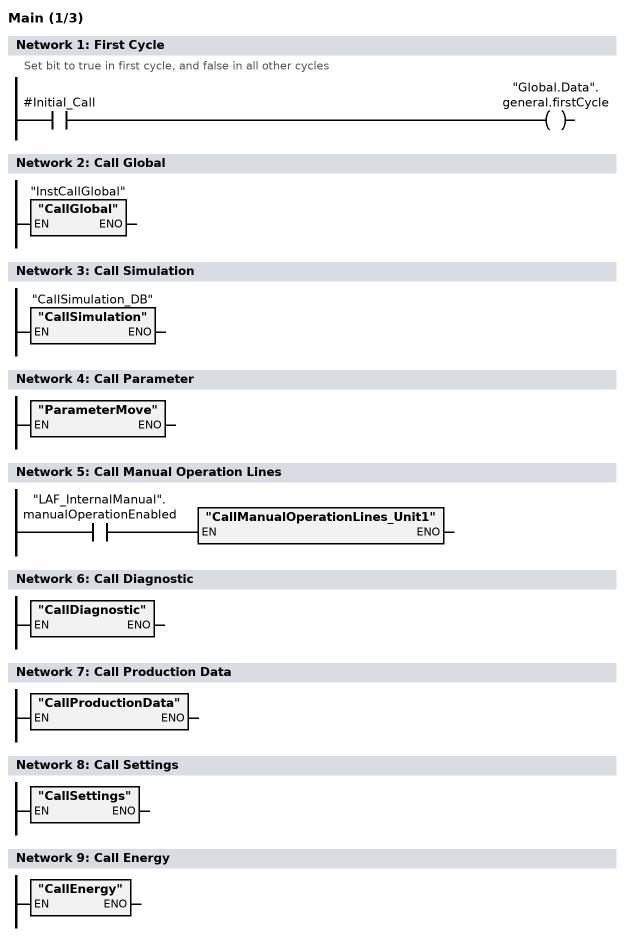
   RUNG wire#powerrail
      Contact( #Initial_Call )
      Coil( "Global.Data".general.firstCycle )
   END_RUNG
   // the same network as SCL:
   "Global.Data".general.firstCycle := #Initial_Call;
END_REGION

REGION Network 2: Call Global
   RUNG wire#powerrail
      "InstCallGlobal"()
   END_RUNG
   // the same network as SCL:
   "InstCallGlobal"();   // "CallGlobal"
END_REGION

REGION Network 3: Call Simulation
   RUNG wire#powerrail
      "CallSimulation_DB"()
   END_RUNG
   // the same network as SCL:
   "CallSimulation_DB"();   // "CallSimulation"
END_REGION

REGION Network 4: Call Parameter
   RUNG wire#powerrail
      "ParameterMove"()
   END_RUNG
   // the same network as SCL:
   "ParameterMove"();
END_REGION

REGION Network 5: Call Manual Operation Lines
   RUNG wire#powerrail
      Contact( "LAF_InternalManual".manualOperationEnabled )
      "CallManualOperationLines_Unit1"()
   END_RUNG
   // the same network as SCL:
   IF "LAF_InternalManual".manualOperationEnabled THEN "CallManualOperationLines_Unit1"(); END_IF;
END_REGION

REGION Network 6: Call Diagnostic
   RUNG wire#powerrail
      "CallDiagnostic"()
   END_RUNG
   // the same network as SCL:
   "CallDiagnostic"();
END_REGION

REGION Network 7: Call Production Data
   RUNG wire#powerrail
      "CallProductionData"()
   END_RUNG
   // the same network as SCL:
   "CallProductionData"();
END_REGION

REGION Network 8: Call Settings
   RUNG wire#powerrail
      "CallSettings"()
   END_RUNG
   // the same network as SCL:
   "CallSettings"();
END_REGION

REGION Network 9: Call Energy
   RUNG wire#powerrail
      "CallEnergy"()
   END_RUNG
   // the same network as SCL:
   "CallEnergy"();
END_REGION

REGION Network 10: HMI SpecialFuction Button Control
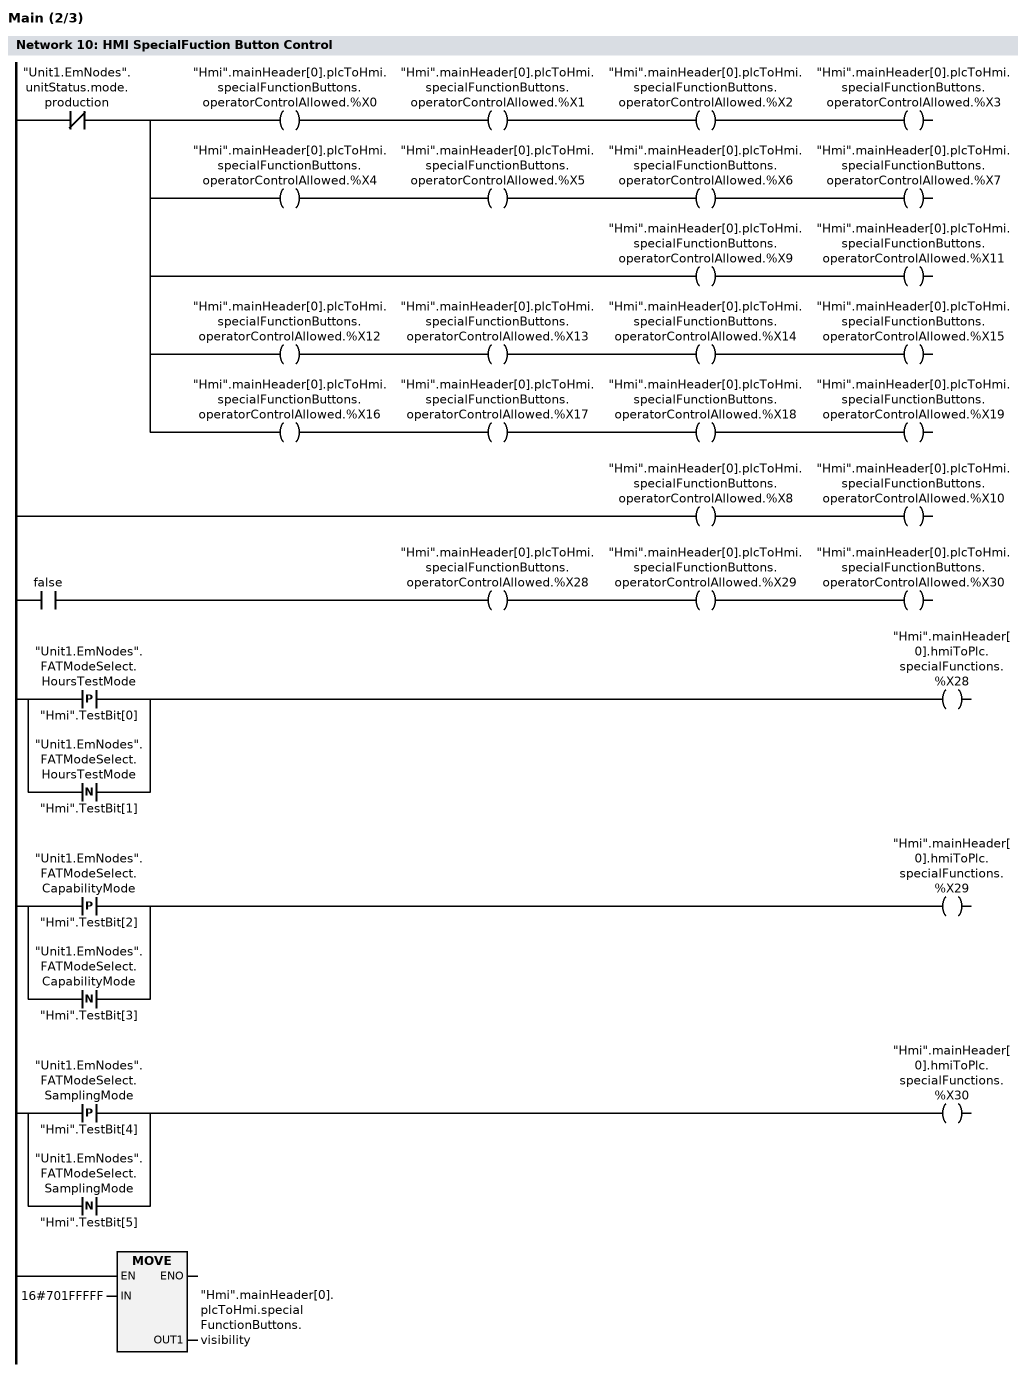
   RUNG wire#powerrail
      I_Contact( "Unit1.EmNodes".unitStatus.mode.production )
      wire#w1
      Coil( "Hmi".mainHeader[0].plcToHmi.specialFunctionButtons.operatorControlAllowed.%X0 )
      Coil( "Hmi".mainHeader[0].plcToHmi.specialFunctionButtons.operatorControlAllowed.%X1 )
      Coil( "Hmi".mainHeader[0].plcToHmi.specialFunctionButtons.operatorControlAllowed.%X2 )
      Coil( "Hmi".mainHeader[0].plcToHmi.specialFunctionButtons.operatorControlAllowed.%X3 )
   END_RUNG
   RUNG wire#w1
      Coil( "Hmi".mainHeader[0].plcToHmi.specialFunctionButtons.operatorControlAllowed.%X4 )
      Coil( "Hmi".mainHeader[0].plcToHmi.specialFunctionButtons.operatorControlAllowed.%X5 )
      Coil( "Hmi".mainHeader[0].plcToHmi.specialFunctionButtons.operatorControlAllowed.%X6 )
      Coil( "Hmi".mainHeader[0].plcToHmi.specialFunctionButtons.operatorControlAllowed.%X7 )
   END_RUNG
   RUNG wire#w1
      Coil( "Hmi".mainHeader[0].plcToHmi.specialFunctionButtons.operatorControlAllowed.%X9 )
      Coil( "Hmi".mainHeader[0].plcToHmi.specialFunctionButtons.operatorControlAllowed.%X11 )
   END_RUNG
   RUNG wire#w1
      Coil( "Hmi".mainHeader[0].plcToHmi.specialFunctionButtons.operatorControlAllowed.%X12 )
      Coil( "Hmi".mainHeader[0].plcToHmi.specialFunctionButtons.operatorControlAllowed.%X13 )
      Coil( "Hmi".mainHeader[0].plcToHmi.specialFunctionButtons.operatorControlAllowed.%X14 )
      Coil( "Hmi".mainHeader[0].plcToHmi.specialFunctionButtons.operatorControlAllowed.%X15 )
   END_RUNG
   RUNG wire#w1
      Coil( "Hmi".mainHeader[0].plcToHmi.specialFunctionButtons.operatorControlAllowed.%X16 )
      Coil( "Hmi".mainHeader[0].plcToHmi.specialFunctionButtons.operatorControlAllowed.%X17 )
      Coil( "Hmi".mainHeader[0].plcToHmi.specialFunctionButtons.operatorControlAllowed.%X18 )
      Coil( "Hmi".mainHeader[0].plcToHmi.specialFunctionButtons.operatorControlAllowed.%X19 )
   END_RUNG
   RUNG wire#powerrail
      Coil( "Hmi".mainHeader[0].plcToHmi.specialFunctionButtons.operatorControlAllowed.%X8 )
      Coil( "Hmi".mainHeader[0].plcToHmi.specialFunctionButtons.operatorControlAllowed.%X10 )
   END_RUNG
   RUNG wire#powerrail
      Contact( false )
      Coil( "Hmi".mainHeader[0].plcToHmi.specialFunctionButtons.operatorControlAllowed.%X28 )
      Coil( "Hmi".mainHeader[0].plcToHmi.specialFunctionButtons.operatorControlAllowed.%X29 )
      Coil( "Hmi".mainHeader[0].plcToHmi.specialFunctionButtons.operatorControlAllowed.%X30 )
   END_RUNG
   RUNG wire#powerrail
      P_Contact(operand := "Unit1.EmNodes".FATModeSelect.HoursTestMode, bit := "Hmi".TestBit[0])
      wire#w2
      Coil( "Hmi".mainHeader[0].hmiToPlc.specialFunctions.%X28 )
   END_RUNG
   RUNG wire#powerrail
      N_Contact(operand := "Unit1.EmNodes".FATModeSelect.HoursTestMode, bit := "Hmi".TestBit[1])
   END_RUNG wire#w2
   RUNG wire#powerrail
      P_Contact(operand := "Unit1.EmNodes".FATModeSelect.CapabilityMode, bit := "Hmi".TestBit[2])
      wire#w3
      Coil( "Hmi".mainHeader[0].hmiToPlc.specialFunctions.%X29 )
   END_RUNG
   RUNG wire#powerrail
      N_Contact(operand := "Unit1.EmNodes".FATModeSelect.CapabilityMode, bit := "Hmi".TestBit[3])
   END_RUNG wire#w3
   RUNG wire#powerrail
      P_Contact(operand := "Unit1.EmNodes".FATModeSelect.SamplingMode, bit := "Hmi".TestBit[4])
      wire#w4
      Coil( "Hmi".mainHeader[0].hmiToPlc.specialFunctions.%X30 )
   END_RUNG
   RUNG wire#powerrail
      N_Contact(operand := "Unit1.EmNodes".FATModeSelect.SamplingMode, bit := "Hmi".TestBit[5])
   END_RUNG wire#w4
   RUNG wire#powerrail
      Move(in := 16#701FFFFF, out1 => "Hmi".mainHeader[0].plcToHmi.specialFunctionButtons.visibility)
   END_RUNG
   // the same network as SCL:
   "Hmi".mainHeader[0].plcToHmi.specialFunctionButtons.operatorControlAllowed.%X0 := NOT "Unit1.EmNodes".unitStatus.mode.production;
   "Hmi".mainHeader[0].plcToHmi.specialFunctionButtons.operatorControlAllowed.%X1 := NOT "Unit1.EmNodes".unitStatus.mode.production;
   "Hmi".mainHeader[0].plcToHmi.specialFunctionButtons.operatorControlAllowed.%X2 := NOT "Unit1.EmNodes".unitStatus.mode.production;
   "Hmi".mainHeader[0].plcToHmi.specialFunctionButtons.operatorControlAllowed.%X3 := NOT "Unit1.EmNodes".unitStatus.mode.production;
   "Hmi".mainHeader[0].plcToHmi.specialFunctionButtons.operatorControlAllowed.%X4 := NOT "Unit1.EmNodes".unitStatus.mode.production;
   "Hmi".mainHeader[0].plcToHmi.specialFunctionButtons.operatorControlAllowed.%X5 := NOT "Unit1.EmNodes".unitStatus.mode.production;
   "Hmi".mainHeader[0].plcToHmi.specialFunctionButtons.operatorControlAllowed.%X6 := NOT "Unit1.EmNodes".unitStatus.mode.production;
   "Hmi".mainHeader[0].plcToHmi.specialFunctionButtons.operatorControlAllowed.%X7 := NOT "Unit1.EmNodes".unitStatus.mode.production;
   "Hmi".mainHeader[0].plcToHmi.specialFunctionButtons.operatorControlAllowed.%X9 := NOT "Unit1.EmNodes".unitStatus.mode.production;
   "Hmi".mainHeader[0].plcToHmi.specialFunctionButtons.operatorControlAllowed.%X11 := NOT "Unit1.EmNodes".unitStatus.mode.production;
   "Hmi".mainHeader[0].plcToHmi.specialFunctionButtons.operatorControlAllowed.%X12 := NOT "Unit1.EmNodes".unitStatus.mode.production;
   "Hmi".mainHeader[0].plcToHmi.specialFunctionButtons.operatorControlAllowed.%X13 := NOT "Unit1.EmNodes".unitStatus.mode.production;
   "Hmi".mainHeader[0].plcToHmi.specialFunctionButtons.operatorControlAllowed.%X14 := NOT "Unit1.EmNodes".unitStatus.mode.production;
   "Hmi".mainHeader[0].plcToHmi.specialFunctionButtons.operatorControlAllowed.%X15 := NOT "Unit1.EmNodes".unitStatus.mode.production;
   "Hmi".mainHeader[0].plcToHmi.specialFunctionButtons.operatorControlAllowed.%X16 := NOT "Unit1.EmNodes".unitStatus.mode.production;
   "Hmi".mainHeader[0].plcToHmi.specialFunctionButtons.operatorControlAllowed.%X17 := NOT "Unit1.EmNodes".unitStatus.mode.production;
   "Hmi".mainHeader[0].plcToHmi.specialFunctionButtons.operatorControlAllowed.%X18 := NOT "Unit1.EmNodes".unitStatus.mode.production;
   "Hmi".mainHeader[0].plcToHmi.specialFunctionButtons.operatorControlAllowed.%X19 := NOT "Unit1.EmNodes".unitStatus.mode.production;
   "Hmi".mainHeader[0].plcToHmi.specialFunctionButtons.operatorControlAllowed.%X8 := TRUE;
   "Hmi".mainHeader[0].plcToHmi.specialFunctionButtons.operatorControlAllowed.%X10 := TRUE;
   "Hmi".mainHeader[0].plcToHmi.specialFunctionButtons.operatorControlAllowed.%X28 := false;
   "Hmi".mainHeader[0].plcToHmi.specialFunctionButtons.operatorControlAllowed.%X29 := false;
   "Hmi".mainHeader[0].plcToHmi.specialFunctionButtons.operatorControlAllowed.%X30 := false;
   #_w1 := "Unit1.EmNodes".FATModeSelect.HoursTestMode AND NOT "Hmi".TestBit[0];   // rising edge of "Unit1.EmNodes".FATModeSelect.HoursTestMode
   "Hmi".TestBit[0] := "Unit1.EmNodes".FATModeSelect.HoursTestMode;
   #_w2 := NOT "Unit1.EmNodes".FATModeSelect.HoursTestMode AND "Hmi".TestBit[1];   // falling edge of "Unit1.EmNodes".FATModeSelect.HoursTestMode
   "Hmi".TestBit[1] := "Unit1.EmNodes".FATModeSelect.HoursTestMode;
   "Hmi".mainHeader[0].hmiToPlc.specialFunctions.%X28 := #_w1 OR #_w2;
   #_w3 := "Unit1.EmNodes".FATModeSelect.CapabilityMode AND NOT "Hmi".TestBit[2];   // rising edge of "Unit1.EmNodes".FATModeSelect.CapabilityMode
   "Hmi".TestBit[2] := "Unit1.EmNodes".FATModeSelect.CapabilityMode;
   #_w4 := NOT "Unit1.EmNodes".FATModeSelect.CapabilityMode AND "Hmi".TestBit[3];   // falling edge of "Unit1.EmNodes".FATModeSelect.CapabilityMode
   "Hmi".TestBit[3] := "Unit1.EmNodes".FATModeSelect.CapabilityMode;
   "Hmi".mainHeader[0].hmiToPlc.specialFunctions.%X29 := #_w3 OR #_w4;
   #_w5 := "Unit1.EmNodes".FATModeSelect.SamplingMode AND NOT "Hmi".TestBit[4];   // rising edge of "Unit1.EmNodes".FATModeSelect.SamplingMode
   "Hmi".TestBit[4] := "Unit1.EmNodes".FATModeSelect.SamplingMode;
   #_w6 := NOT "Unit1.EmNodes".FATModeSelect.SamplingMode AND "Hmi".TestBit[5];   // falling edge of "Unit1.EmNodes".FATModeSelect.SamplingMode
   "Hmi".TestBit[5] := "Unit1.EmNodes".FATModeSelect.SamplingMode;
   "Hmi".mainHeader[0].hmiToPlc.specialFunctions.%X30 := #_w5 OR #_w6;
   "Hmi".mainHeader[0].plcToHmi.specialFunctionButtons.visibility := 16#701FFFFF;
END_REGION

REGION Network 11
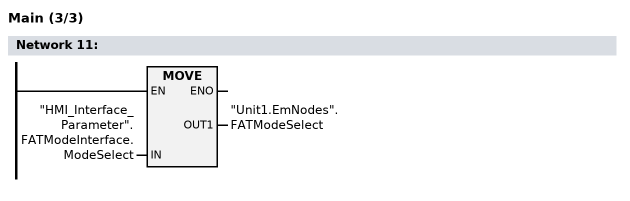
   RUNG wire#powerrail
      Move(in := "HMI_Interface_Parameter".FATModeInterface.ModeSelect, out1 => "Unit1.EmNodes".FATModeSelect)
   END_RUNG
   // the same network as SCL:
   "Unit1.EmNodes".FATModeSelect := "HMI_Interface_Parameter".FATModeInterface.ModeSelect;
END_REGION
END_ORGANIZATION_BLOCK

FUNCTION_BLOCK "CallGlobal"   // FB48, LAD
TITLE = CallGlobal
// All blocks that provide data to the DB Global.Data are called here. That includes blocks to generate system data as well as blocks that connect handle multiple HMIs.
// stored: IsIECCheckEnabled true, MemoryReserve 100, SetENOAutomatically true
   VAR
      statClockSysMemOld { ExternalWritable := 'False'} : Byte;   // Alter Wert Systeminformationsspeicher auswertung / Old value system memory evaluation
      statTonTimer : Array[0..1] of IEC_TIMER;
      instLAF_PowerOnOff { ExternalWritable := 'False'} : "LAF_PowerOnOff";
      instLAF_HmiHeaderManager { ExternalWritable := 'False'} : "LAF_HmiHeaderManager";
      instLAF_ClockGen { ExternalWritable := 'False'} : "LAF_ClockGenerator";
      instLSNTP_Server { ExternalWritable := 'False'} : "LSNTP_Server";
      instRemoteAccess { ExternalWritable := 'False'} : "LRemoteAccess_MobilePanelMonitor";
      statPulse : Array[0..99] of Bool;
   END_VAR
   VAR_TEMP
      tempIndex : DInt;   // Temp variable for for loop
      tempAcknowledge : Bool;   // Summarized acknowledge command
      tempPowerOff : Bool;   // Summarized power off command
      tempPowerOn : Bool;   // Summarized power on command
      tempPowerStatus : Int;   // 0 - Off, 1 - Paused, 2 - On
      tempResultXor : Byte;   // Zwischenergebnis von XOR Anweisung / Interim result of XOR operation
      tempPosPulse : Byte;   // Zwischenergebnis von Pulsauswertung / Interim result puls calculation
   END_VAR
   VAR CONSTANT
      RESET_BUTTON__COULD_BE_ADDED_HERE : Bool := false;   // Placeholder for a potential global reset button
      TRUE : Bool := true;
   END_VAR
   VAR_TEMP   // added for the SCL form of the ladder/FBD networks
      _w1 : Bool;
      _w2 : Bool;
      _w3 : Bool;
   END_VAR
BEGIN

REGION Network 1 (SCL): Summarize HMI commands
   // Read commands for acknowledge, powerOn and powerOff from the different HMI panels and summarize them in temp variables for further logic in this block.
   // Initialize temp variables
   #tempAcknowledge :=
   #tempPowerOff :=
   #tempPowerOn := FALSE;

   // Loop through the HMI panels and summarize the commands
   FOR #tempIndex := 0 TO "NO_OF_PANELS" DO
       #tempAcknowledge := #tempAcknowledge OR "Hmi".mainHeader[#tempIndex].hmiToPlc.acknowledge;
       #tempPowerOff := #tempPowerOff OR "Hmi".mainHeader[#tempIndex].hmiToPlc.powerCommands.%X0;
       #tempPowerOn := #tempPowerOn OR "Hmi".mainHeader[#tempIndex].hmiToPlc.powerCommands.%X1;
   END_FOR;
END_REGION

REGION Network 2: Global Acknowledge
   // The global acknowledge command from the hmi button is assigned to Global.Data.general.acknowledge: This bit it forwarded to all underlaying modules
   // If a hard-wired global reset button exists, it can
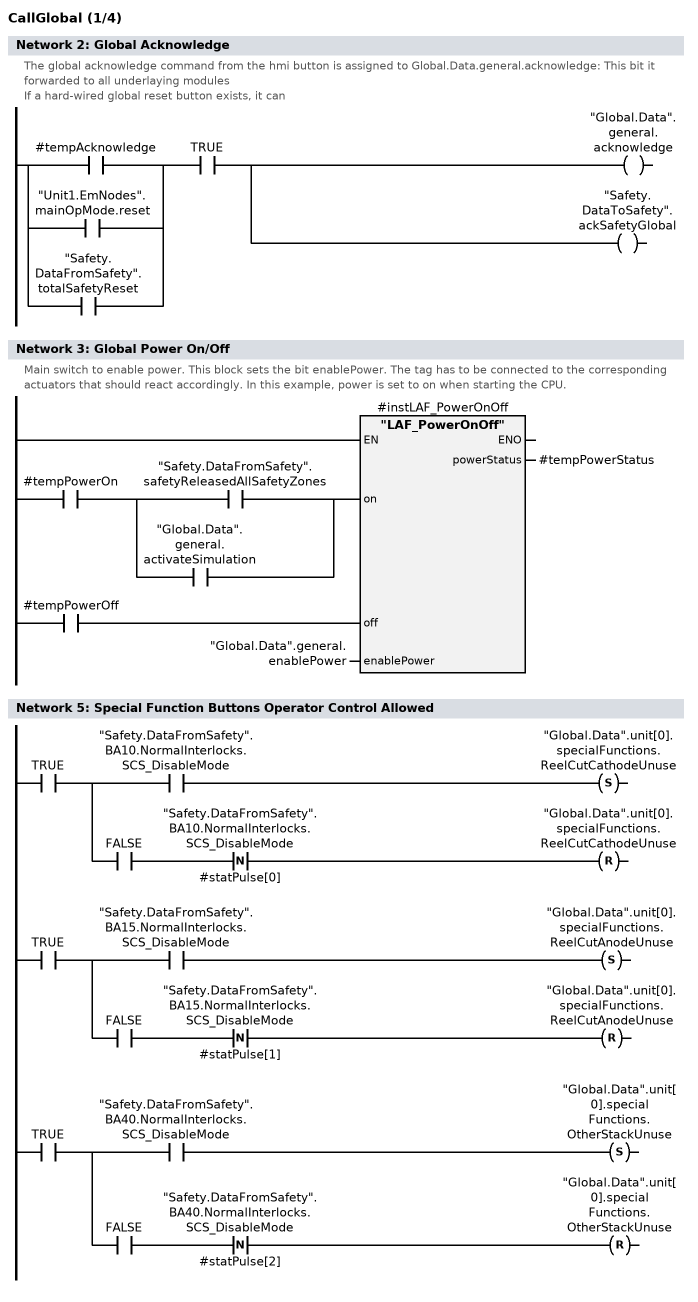
   RUNG wire#powerrail
      Contact( #tempAcknowledge )
      wire#w1
      Contact( TRUE )
      wire#w2
      Coil( "Global.Data".general.acknowledge )
   END_RUNG
   RUNG wire#powerrail
      Contact( "Unit1.EmNodes".mainOpMode.reset )
   END_RUNG wire#w1
   RUNG wire#powerrail
      Contact( "Safety.DataFromSafety".totalSafetyReset )
   END_RUNG wire#w1
   RUNG wire#w2
      Coil( "Safety.DataToSafety".ackSafetyGlobal )
   END_RUNG
   // the same network as SCL:
   "Global.Data".general.acknowledge := (#tempAcknowledge OR "Unit1.EmNodes".mainOpMode.reset OR "Safety.DataFromSafety".totalSafetyReset) AND TRUE;
   "Safety.DataToSafety".ackSafetyGlobal := "Global.Data".general.acknowledge;
END_REGION

REGION Network 3: Global Power On/Off
   // Main switch to enable power. This block sets the bit enablePower. The tag has to be connected to the corresponding actuators that should react accordingly. In this example, power is set to on when starting the CPU.
   RUNG wire#powerrail
      #instLAF_PowerOnOff(on := wire#w2, off := wire#w3, enablePower := "Global.Data".general.enablePower, powerStatus => #tempPowerStatus)
   END_RUNG
   RUNG wire#powerrail
      Contact( #tempPowerOn )
      wire#w1
      Contact( "Safety.DataFromSafety".safetyReleasedAllSafetyZones )
   END_RUNG wire#w2
   RUNG wire#w1
      Contact( "Global.Data".general.activateSimulation )
   END_RUNG wire#w2
   RUNG wire#powerrail
      Contact( #tempPowerOff )
   END_RUNG wire#w3
   // the same network as SCL:
   #instLAF_PowerOnOff(on := #tempPowerOn AND ("Safety.DataFromSafety".safetyReleasedAllSafetyZones OR "Global.Data".general.activateSimulation),   // "LAF_PowerOnOff"
                       off := #tempPowerOff,
                       enablePower := "Global.Data".general.enablePower,
                       powerStatus => #tempPowerStatus);
END_REGION

REGION Network 4 (SCL): Write power status to HMI panels
   // Write power status back to all connected HMI panels
   // Loop through the panels and set the power status
   FOR #tempIndex := 0 TO "NO_OF_PANELS" DO
       "Hmi".mainHeader[#tempIndex].plcToHmi.powerStatus := #tempPowerStatus;
   END_FOR;
END_REGION

REGION Network 5: Special Function Buttons Operator Control Allowed
   RUNG wire#powerrail
      Contact( TRUE )
      wire#w1
      Contact( "Safety.DataFromSafety".BA10.NormalInterlocks.SCS_DisableMode )
      S_Coil( "Global.Data".unit[0].specialFunctions.ReelCutCathodeUnuse )
   END_RUNG
   RUNG wire#w1
      Contact( FALSE )
      N_Contact(operand := "Safety.DataFromSafety".BA10.NormalInterlocks.SCS_DisableMode, bit := #statPulse[0])
      R_Coil( "Global.Data".unit[0].specialFunctions.ReelCutCathodeUnuse )
   END_RUNG
   RUNG wire#powerrail
      Contact( TRUE )
      wire#w2
      Contact( "Safety.DataFromSafety".BA15.NormalInterlocks.SCS_DisableMode )
      S_Coil( "Global.Data".unit[0].specialFunctions.ReelCutAnodeUnuse )
   END_RUNG
   RUNG wire#w2
      Contact( FALSE )
      N_Contact(operand := "Safety.DataFromSafety".BA15.NormalInterlocks.SCS_DisableMode, bit := #statPulse[1])
      R_Coil( "Global.Data".unit[0].specialFunctions.ReelCutAnodeUnuse )
   END_RUNG
   RUNG wire#powerrail
      Contact( TRUE )
      wire#w3
      Contact( "Safety.DataFromSafety".BA40.NormalInterlocks.SCS_DisableMode )
      S_Coil( "Global.Data".unit[0].specialFunctions.OtherStackUnuse )
   END_RUNG
   RUNG wire#w3
      Contact( FALSE )
      N_Contact(operand := "Safety.DataFromSafety".BA40.NormalInterlocks.SCS_DisableMode, bit := #statPulse[2])
      R_Coil( "Global.Data".unit[0].specialFunctions.OtherStackUnuse )
   END_RUNG
   // the same network as SCL:
   IF TRUE AND "Safety.DataFromSafety".BA10.NormalInterlocks.SCS_DisableMode THEN
       "Global.Data".unit[0].specialFunctions.ReelCutCathodeUnuse := TRUE;
   END_IF;
   #_w1 := TRUE AND FALSE AND NOT "Safety.DataFromSafety".BA10.NormalInterlocks.SCS_DisableMode AND #statPulse[0];   // falling edge of "Safety.DataFromSafety".BA10.NormalInterlocks.SCS_DisableMode
   #statPulse[0] := "Safety.DataFromSafety".BA10.NormalInterlocks.SCS_DisableMode;
   IF #_w1 THEN "Global.Data".unit[0].specialFunctions.ReelCutCathodeUnuse := FALSE; END_IF;
   IF TRUE AND "Safety.DataFromSafety".BA15.NormalInterlocks.SCS_DisableMode THEN
       "Global.Data".unit[0].specialFunctions.ReelCutAnodeUnuse := TRUE;
   END_IF;
   #_w2 := TRUE AND FALSE AND NOT "Safety.DataFromSafety".BA15.NormalInterlocks.SCS_DisableMode AND #statPulse[1];   // falling edge of "Safety.DataFromSafety".BA15.NormalInterlocks.SCS_DisableMode
   #statPulse[1] := "Safety.DataFromSafety".BA15.NormalInterlocks.SCS_DisableMode;
   IF #_w2 THEN "Global.Data".unit[0].specialFunctions.ReelCutAnodeUnuse := FALSE; END_IF;
   IF TRUE AND "Safety.DataFromSafety".BA40.NormalInterlocks.SCS_DisableMode THEN
       "Global.Data".unit[0].specialFunctions.OtherStackUnuse := TRUE;
   END_IF;
   #_w3 := TRUE AND FALSE AND NOT "Safety.DataFromSafety".BA40.NormalInterlocks.SCS_DisableMode AND #statPulse[2];   // falling edge of "Safety.DataFromSafety".BA40.NormalInterlocks.SCS_DisableMode
   #statPulse[2] := "Safety.DataFromSafety".BA40.NormalInterlocks.SCS_DisableMode;
   IF #_w3 THEN "Global.Data".unit[0].specialFunctions.OtherStackUnuse := FALSE; END_IF;
END_REGION

REGION Network 6: HMI Control Header
   // Read the input from the control header in the HMI an distribute information to the according units. Vice versa, summarize the unit information and provide it to the control header to display e.g. the modes and states.
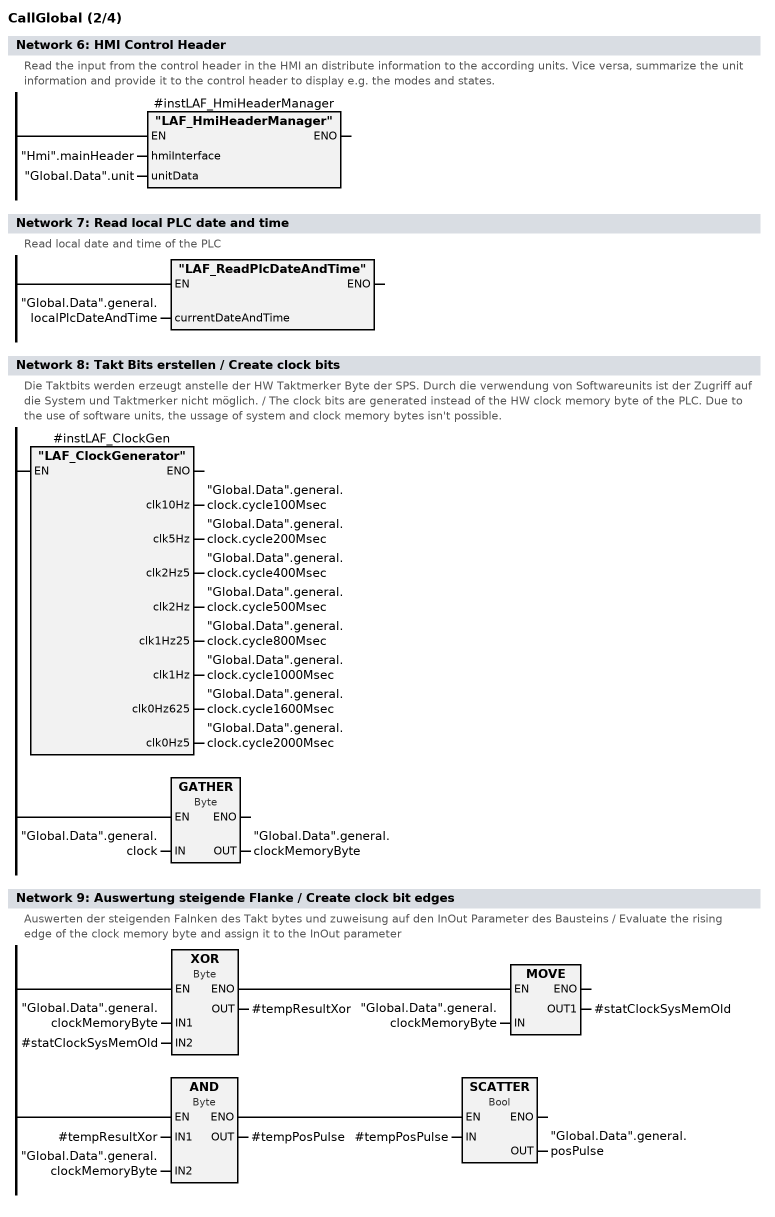
   RUNG wire#powerrail
      #instLAF_HmiHeaderManager(hmiInterface := "Hmi".mainHeader, unitData := "Global.Data".unit)
   END_RUNG
   // the same network as SCL:
   #instLAF_HmiHeaderManager(hmiInterface := "Hmi".mainHeader, unitData := "Global.Data".unit);   // "LAF_HmiHeaderManager"
END_REGION

REGION Network 7: Read local PLC date and time
   // Read local date and time of the PLC
   RUNG wire#powerrail
      "LAF_ReadPlcDateAndTime"(currentDateAndTime := "Global.Data".general.localPlcDateAndTime)
   END_RUNG
   // the same network as SCL:
   "LAF_ReadPlcDateAndTime"(currentDateAndTime := "Global.Data".general.localPlcDateAndTime);
END_REGION

REGION Network 8: Takt Bits erstellen / Create clock bits
   // Die Taktbits werden erzeugt anstelle der HW Taktmerker Byte der SPS. Durch die verwendung von Softwareunits ist der Zugriff auf die System und Taktmerker nicht möglich. / The clock bits are generated instead of the HW clock memory byte of the PLC. Due to the use of software units, the ussage of system and clock memory bytes isn't possible.
   RUNG wire#powerrail
      #instLAF_ClockGen(clk10Hz => "Global.Data".general.clock.cycle100Msec, clk5Hz => "Global.Data".general.clock.cycle200Msec, clk2Hz5 => "Global.Data".general.clock.cycle400Msec, clk2Hz => "Global.Data".general.clock.cycle500Msec, clk1Hz25 => "Global.Data".general.clock.cycle800Msec, clk1Hz => "Global.Data".general.clock.cycle1000Msec, clk0Hz625 => "Global.Data".general.clock.cycle1600Msec, clk0Hz5 => "Global.Data".general.clock.cycle2000Msec)
   END_RUNG
   RUNG wire#powerrail
      { S7_Templates := "[dest_type := Byte, src_type := Bool]" } GATHER(IN := "Global.Data".general.clock, OUT => "Global.Data".general.clockMemoryByte)
   END_RUNG
   // the same network as SCL:
   #instLAF_ClockGen(clk10Hz => "Global.Data".general.clock.cycle100Msec,   // "LAF_ClockGenerator"
                     clk5Hz => "Global.Data".general.clock.cycle200Msec,
                     clk2Hz5 => "Global.Data".general.clock.cycle400Msec,
                     clk2Hz => "Global.Data".general.clock.cycle500Msec,
                     clk1Hz25 => "Global.Data".general.clock.cycle800Msec,
                     clk1Hz => "Global.Data".general.clock.cycle1000Msec,
                     clk0Hz625 => "Global.Data".general.clock.cycle1600Msec,
                     clk0Hz5 => "Global.Data".general.clock.cycle2000Msec);
   GATHER(IN := "Global.Data".general.clock, OUT => "Global.Data".general.clockMemoryByte);
END_REGION

REGION Network 9: Auswertung steigende Flanke / Create clock bit edges
   // Auswerten der steigenden Falnken des Takt bytes und zuweisung auf den InOut Parameter des Bausteins / Evaluate the rising edge of the clock memory byte and assign it to the InOut parameter
   #tempResultXor := "Global.Data".general.clockMemoryByte XOR #statClockSysMemOld;
   #statClockSysMemOld := "Global.Data".general.clockMemoryByte;
   #tempPosPulse := #tempResultXor AND "Global.Data".general.clockMemoryByte;
   SCATTER(IN := #tempPosPulse, OUT => "Global.Data".general.posPulse);
END_REGION

REGION Network 10: Time Synchronisation (NTP)
   // With the LSNTP_Server block, the NTP server will be enabled on S7 PLC, to wich the NTP client (e.g. Panel), can synchronize their data and time.
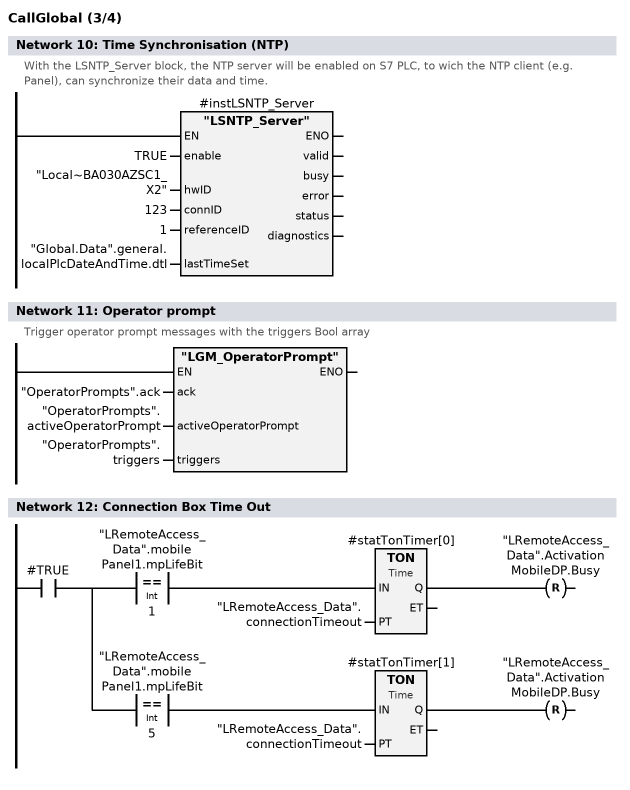
   RUNG wire#powerrail
      #instLSNTP_Server(enable := TRUE, hwID := "Local~BA030AZSC1_X2", connID := 123, referenceID := 1, lastTimeSet := "Global.Data".general.localPlcDateAndTime.dtl, valid =>, busy =>, error =>, status =>, diagnostics =>)
   END_RUNG
   // the same network as SCL:
   #instLSNTP_Server(enable := TRUE,   // "LSNTP_Server"
                     hwID := "Local~BA030AZSC1_X2",
                     connID := 123,
                     referenceID := 1,
                     lastTimeSet := "Global.Data".general.localPlcDateAndTime.dtl);
END_REGION

REGION Network 11: Operator prompt
   // Trigger operator prompt messages with the triggers Bool array
   RUNG wire#powerrail
      "LGM_OperatorPrompt"(ack := "OperatorPrompts".ack, activeOperatorPrompt := "OperatorPrompts".activeOperatorPrompt, triggers := "OperatorPrompts".triggers)
   END_RUNG
   // the same network as SCL:
   "LGM_OperatorPrompt"(ack := "OperatorPrompts".ack,
                        activeOperatorPrompt := "OperatorPrompts".activeOperatorPrompt,
                        triggers := "OperatorPrompts".triggers);
END_REGION

REGION Network 12: Connection Box Time Out
   RUNG wire#powerrail
      Contact( #TRUE )
      wire#w1
      { S7_Templates := "SrcType := Int" } EQ_Contact(in1 := "LRemoteAccess_Data".mobilePanel1.mpLifeBit, in2 := 1)
      { S7_Templates := "time_type := Time" } #statTonTimer[0].TON(pt := "LRemoteAccess_Data".connectionTimeout, et =>)
      R_Coil( "LRemoteAccess_Data".ActivationMobileDP.Busy )
   END_RUNG
   RUNG wire#w1
      { S7_Templates := "SrcType := Int" } EQ_Contact(in1 := "LRemoteAccess_Data".mobilePanel1.mpLifeBit, in2 := 5)
      { S7_Templates := "time_type := Time" } #statTonTimer[1].TON(pt := "LRemoteAccess_Data".connectionTimeout, et =>)
      R_Coil( "LRemoteAccess_Data".ActivationMobileDP.Busy )
   END_RUNG
   // the same network as SCL:
   #statTonTimer[0].TON(IN := #TRUE AND ("LRemoteAccess_Data".mobilePanel1.mpLifeBit = 1),
                        PT := "LRemoteAccess_Data".connectionTimeout);
   IF #statTonTimer[0].Q THEN "LRemoteAccess_Data".ActivationMobileDP.Busy := FALSE; END_IF;
   #statTonTimer[1].TON(IN := #TRUE AND ("LRemoteAccess_Data".mobilePanel1.mpLifeBit = 5),
                        PT := "LRemoteAccess_Data".connectionTimeout);
   IF #statTonTimer[1].Q THEN "LRemoteAccess_Data".ActivationMobileDP.Busy := FALSE; END_IF;
END_REGION

REGION Network 13: Connection box is connected
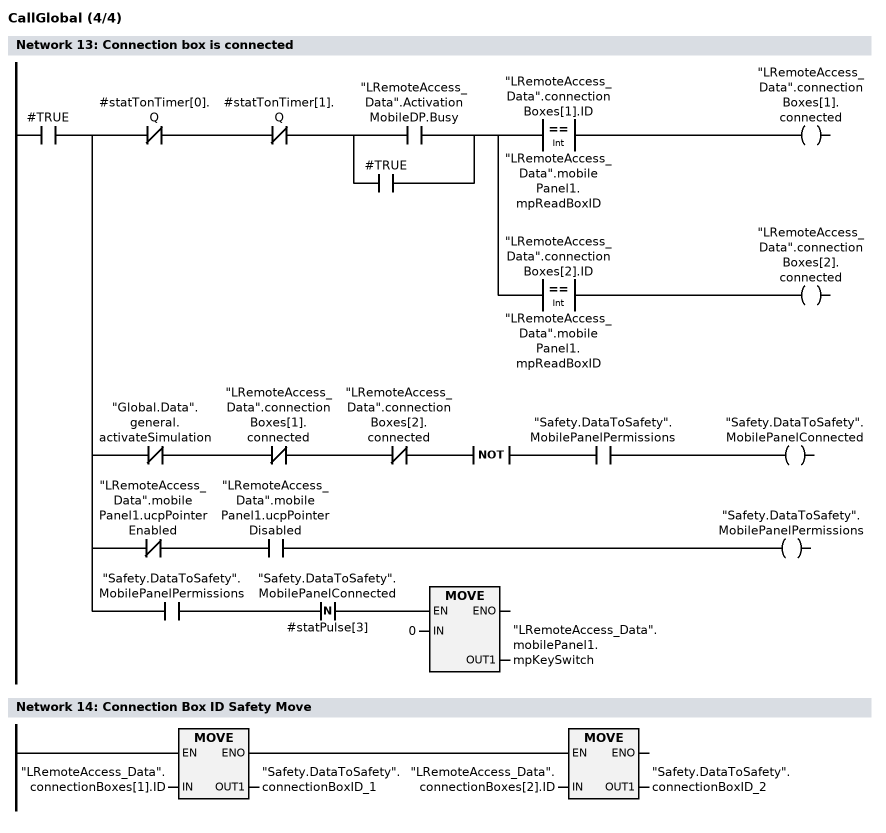
   RUNG wire#powerrail
      Contact( #TRUE )
      wire#w1
      I_Contact( #statTonTimer[0].Q )
      I_Contact( #statTonTimer[1].Q )
      wire#w2
      Contact( "LRemoteAccess_Data".ActivationMobileDP.Busy )
      wire#w3
      { S7_Templates := "SrcType := Int" } EQ_Contact(in1 := "LRemoteAccess_Data".connectionBoxes[1].ID, in2 := "LRemoteAccess_Data".mobilePanel1.mpReadBoxID)
      Coil( "LRemoteAccess_Data".connectionBoxes[1].connected )
   END_RUNG
   RUNG wire#w2
      Contact( #TRUE )
   END_RUNG wire#w3
   RUNG wire#w3
      { S7_Templates := "SrcType := Int" } EQ_Contact(in1 := "LRemoteAccess_Data".connectionBoxes[2].ID, in2 := "LRemoteAccess_Data".mobilePanel1.mpReadBoxID)
      Coil( "LRemoteAccess_Data".connectionBoxes[2].connected )
   END_RUNG
   RUNG wire#w1
      I_Contact( "Global.Data".general.activateSimulation )
      I_Contact( "LRemoteAccess_Data".connectionBoxes[1].connected )
      I_Contact( "LRemoteAccess_Data".connectionBoxes[2].connected )
      Not()
      Contact( "Safety.DataToSafety".MobilePanelPermissions )
      Coil( "Safety.DataToSafety".MobilePanelConnected )
   END_RUNG
   RUNG wire#w1
      I_Contact( "LRemoteAccess_Data".mobilePanel1.ucpPointerEnabled )
      Contact( "LRemoteAccess_Data".mobilePanel1.ucpPointerDisabled )
      Coil( "Safety.DataToSafety".MobilePanelPermissions )
   END_RUNG
   RUNG wire#w1
      Contact( "Safety.DataToSafety".MobilePanelPermissions )
      N_Contact(operand := "Safety.DataToSafety".MobilePanelConnected, bit := #statPulse[3])
      Move(in := 0, out1 => "LRemoteAccess_Data".mobilePanel1.mpKeySwitch)
   END_RUNG
   // the same network as SCL:
   #_w1 := #TRUE AND NOT #statTonTimer[0].Q AND NOT #statTonTimer[1].Q AND ("LRemoteAccess_Data".ActivationMobileDP.Busy OR #TRUE);
   "LRemoteAccess_Data".connectionBoxes[1].connected := #_w1 AND ("LRemoteAccess_Data".connectionBoxes[1].ID = "LRemoteAccess_Data".mobilePanel1.mpReadBoxID);
   "LRemoteAccess_Data".connectionBoxes[2].connected := #_w1 AND ("LRemoteAccess_Data".connectionBoxes[2].ID = "LRemoteAccess_Data".mobilePanel1.mpReadBoxID);
   "Safety.DataToSafety".MobilePanelConnected := NOT (#TRUE AND NOT "Global.Data".general.activateSimulation AND NOT "LRemoteAccess_Data".connectionBoxes[1].connected AND NOT "LRemoteAccess_Data".connectionBoxes[2].connected) AND "Safety.DataToSafety".MobilePanelPermissions;
   "Safety.DataToSafety".MobilePanelPermissions := #TRUE AND NOT "LRemoteAccess_Data".mobilePanel1.ucpPointerEnabled AND "LRemoteAccess_Data".mobilePanel1.ucpPointerDisabled;
   #_w2 := #TRUE AND "Safety.DataToSafety".MobilePanelPermissions AND NOT "Safety.DataToSafety".MobilePanelConnected AND #statPulse[3];   // falling edge of "Safety.DataToSafety".MobilePanelConnected
   #statPulse[3] := "Safety.DataToSafety".MobilePanelConnected;
   IF #_w2 THEN "LRemoteAccess_Data".mobilePanel1.mpKeySwitch := 0; END_IF;
END_REGION

REGION Network 14: Connection Box ID Safety Move
   RUNG wire#powerrail
      Move(in := "LRemoteAccess_Data".connectionBoxes[1].ID, out1 => "Safety.DataToSafety".connectionBoxID_1)
      Move(in := "LRemoteAccess_Data".connectionBoxes[2].ID, out1 => "Safety.DataToSafety".connectionBoxID_2)
   END_RUNG
   // the same network as SCL:
   "Safety.DataToSafety".connectionBoxID_1 := "LRemoteAccess_Data".connectionBoxes[1].ID;
   "Safety.DataToSafety".connectionBoxID_2 := "LRemoteAccess_Data".connectionBoxes[2].ID;
END_REGION
END_FUNCTION_BLOCK

FUNCTION_BLOCK "CallSimulation"   // FB19, LAD
// stored: MemoryReserve 100, SetENOAutomatically false
   VAR
      instSimRotaryAxis { ExternalAccessible := 'False'; ExternalVisible := 'False'; ExternalWritable := 'False'} : Array[0..49] of "LER_SimHmiRotaryAxis";
      Unwindwe1 { S7_SetPoint := 'True'} : "LER_SimHmiRotaryAxis";
      IEC_Timer_0_Instance { S7_SetPoint := 'True'} : TON_TIME;
      "LER_SimAxis+_Axis07_pnp1X" { S7_SetPoint := 'True'} : "LER_SimAxis+";
      "LER_SimAxis+_Axis10_pnp1Z" { S7_SetPoint := 'True'} : "LER_SimAxis+";
      "LER_SimAxis+_Axis8_pnp2X" { S7_SetPoint := 'True'} : "LER_SimAxis+";
      "LER_SimAxis+_Axis13_pnp2Z" { S7_SetPoint := 'True'} : "LER_SimAxis+";
      "LER_SimAxis+_Axis12_pnp1Z" { S7_SetPoint := 'True'} : "LER_SimAxis+";
      "LER_SimAxis+_Axis14_pnp2Z" { S7_SetPoint := 'True'} : "LER_SimAxis+";
      "LER_SimAxis+_Axis34_cutterX" { S7_SetPoint := 'True'} : "LER_SimAxis+";
      "LER_SimAxis+_Axis35_cutterZ" { S7_SetPoint := 'True'} : "LER_SimAxis+";
      "LER_SimAxis-_Axis36_GripperX" { S7_SetPoint := 'True'} : "LER_SimAxis-";
      "LER_SimAxis+_Axis37_gripperZ" { S7_SetPoint := 'True'} : "LER_SimAxis+";
      "LER_SimAxis-_Axis32_StackTableZ" { S7_SetPoint := 'True'} : "LER_SimAxis-";
      "LER_SimAxis+_Axis21_roller" { S7_SetPoint := 'True'} : "LER_SimAxis+";
      "LER_SimAxis+_gripperAxis_C" { S7_SetPoint := 'True'} : "LER_SimAxis+";
      IEC_Timer_1_Instance { S7_SetPoint := 'True'} : TON_TIME;
      "LER_SimAxis+_Axis05_pnp1X" { S7_SetPoint := 'True'} : "LER_SimAxis+";
      "LER_SimAxis+_Axis06_pnp2X" { S7_SetPoint := 'True'} : "LER_SimAxis+";
   END_VAR
   VAR CONSTANT
      FALSE : Bool := FALSE;
      TRUE : Bool := TRUE;
   END_VAR
   VAR_TEMP   // added for the SCL form of the ladder/FBD networks
      _w1 : Bool;
      _w2 : Bool;
      _w3 : Bool;
      _w4 : Bool;
      _w5 : Bool;
      _w6 : Bool;
      _w7 : Bool;
      _w8 : Bool;
   END_VAR
BEGIN

REGION Network 1: SIMIT simulation currently running
   // The input "0.000CC1-KE50_I1.6_SimitRunning" is a life bit from SIMIT, which is always TRUE while SIMIT is running. The following actions are performed in that case:
   // - Simulation button in HMI is not shown when a SIMIT simulation is currently running
   // - Deactivate PLC internal simulation while SIMIT simulation is running
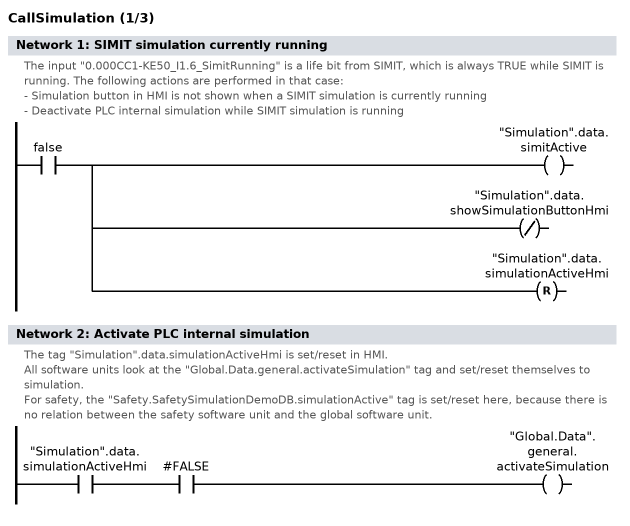
   RUNG wire#powerrail
      Contact( false )
      wire#w1
      Coil( "Simulation".data.simitActive )
   END_RUNG
   RUNG wire#w1
      I_Coil( "Simulation".data.showSimulationButtonHmi )
   END_RUNG
   RUNG wire#w1
      R_Coil( "Simulation".data.simulationActiveHmi )
   END_RUNG
   // the same network as SCL:
   "Simulation".data.simitActive := false;
   "Simulation".data.showSimulationButtonHmi := NOT false;
   IF false THEN "Simulation".data.simulationActiveHmi := FALSE; END_IF;
END_REGION

REGION Network 2: Activate PLC internal simulation
   // The tag "Simulation".data.simulationActiveHmi is set/reset in HMI.
   // 
   // All software units look at the "Global.Data.general.activateSimulation" tag and set/reset themselves to simulation.
   // 
   // For safety, the "Safety.SafetySimulationDemoDB.simulationActive" tag is set/reset here, because there is no relation between the safety software unit and the global software unit.
   RUNG wire#powerrail
      Contact( "Simulation".data.simulationActiveHmi )
      Contact( #FALSE )
      Coil( "Global.Data".general.activateSimulation )
   END_RUNG
   // the same network as SCL:
   "Global.Data".general.activateSimulation := "Simulation".data.simulationActiveHmi AND #FALSE;
END_REGION

REGION Network 3: Simulation Linear Axis
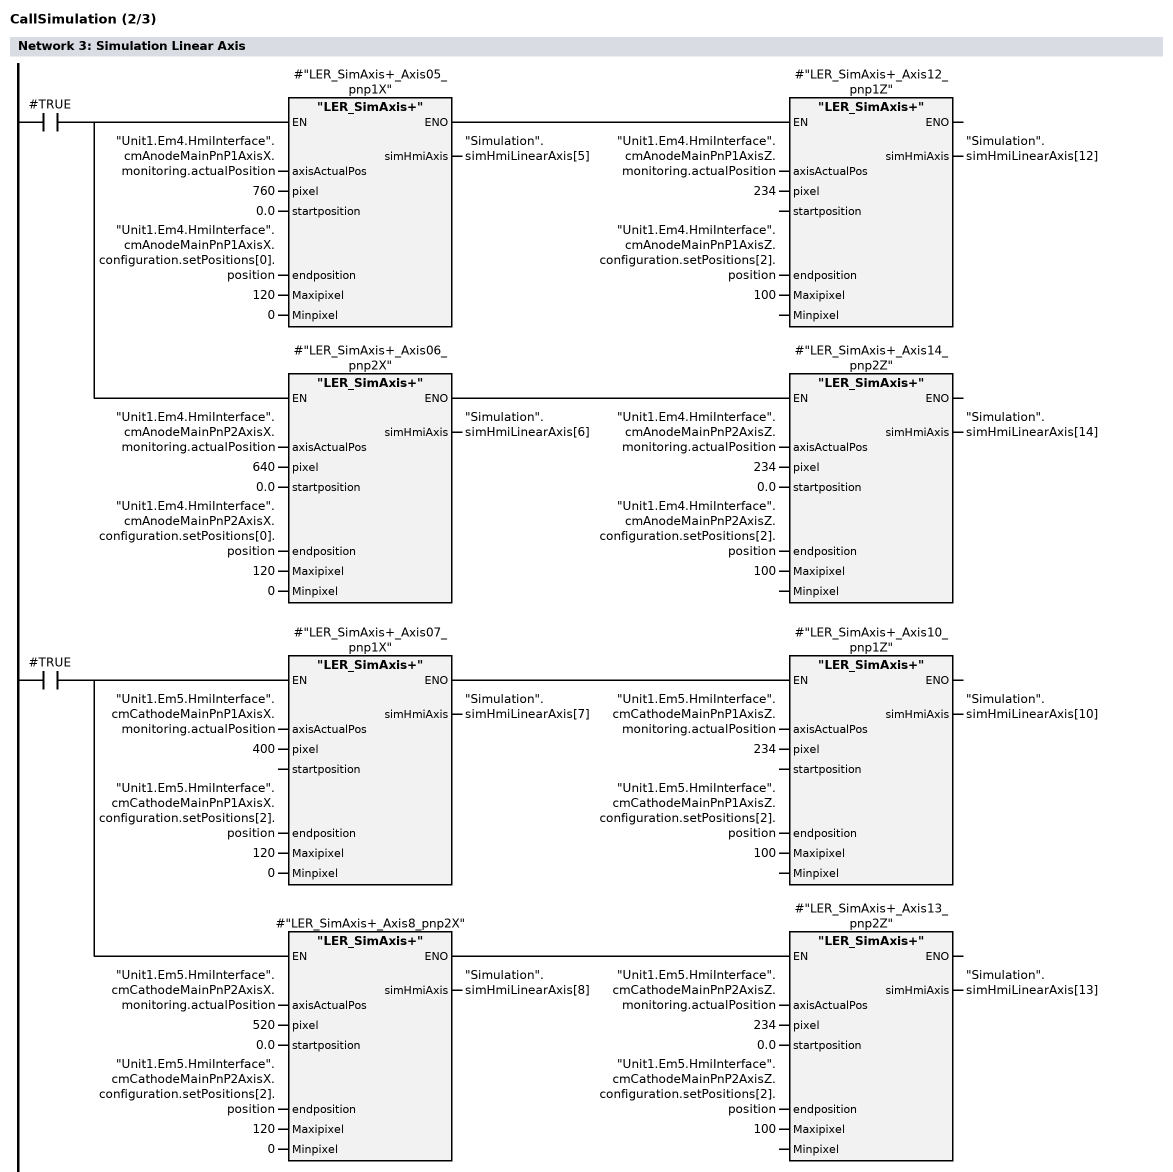
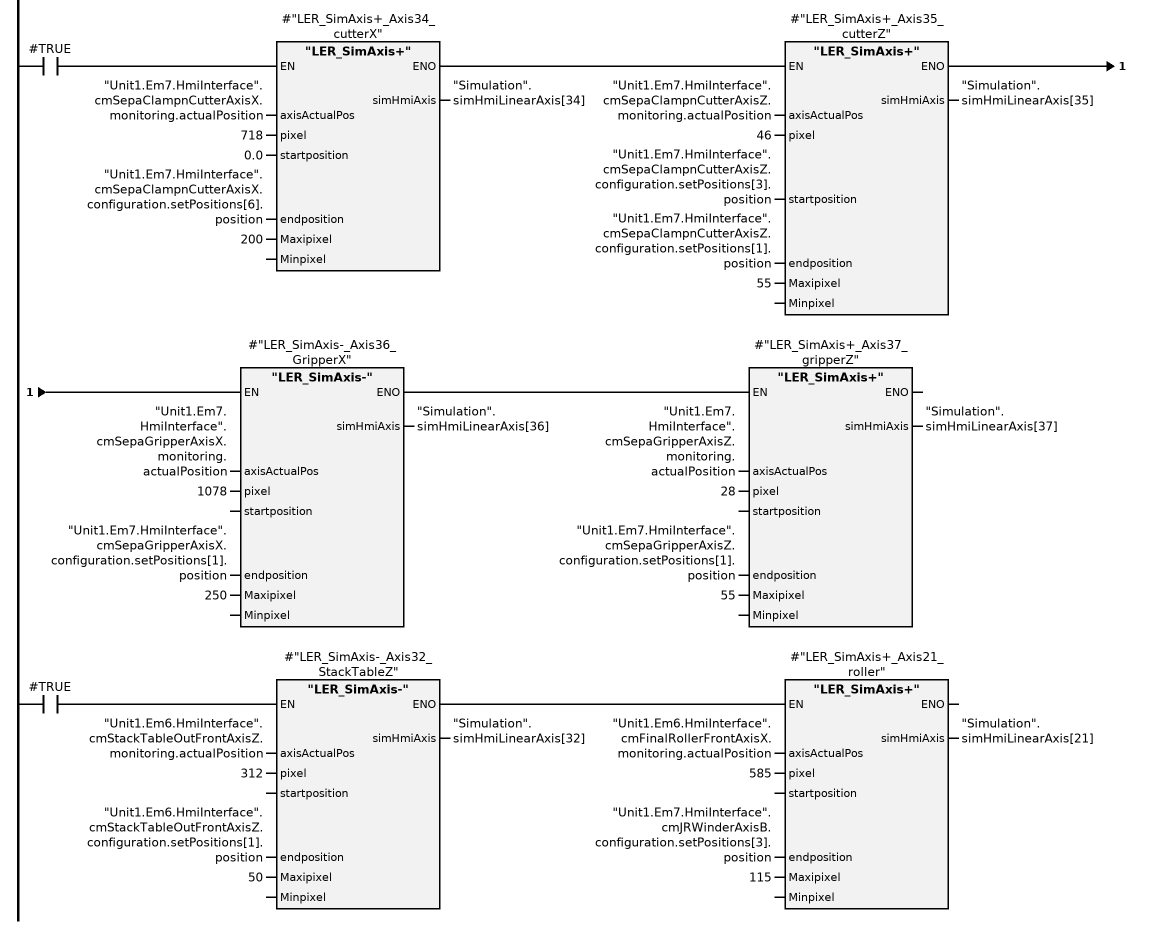
   RUNG wire#powerrail
      Contact( #TRUE )
      wire#w1
      #"LER_SimAxis+_Axis05_pnp1X"(axisActualPos := "Unit1.Em4.HmiInterface".cmAnodeMainPnP1AxisX.monitoring.actualPosition, pixel := 760, startposition := 0.0, endposition := "Unit1.Em4.HmiInterface".cmAnodeMainPnP1AxisX.configuration.setPositions[0].position, Maxipixel := 120, Minpixel := 0, simHmiAxis => "Simulation".simHmiLinearAxis[5])
      #"LER_SimAxis+_Axis12_pnp1Z"(axisActualPos := "Unit1.Em4.HmiInterface".cmAnodeMainPnP1AxisZ.monitoring.actualPosition, pixel := 234, startposition :=, endposition := "Unit1.Em4.HmiInterface".cmAnodeMainPnP1AxisZ.configuration.setPositions[2].position, Maxipixel := 100, Minpixel :=, simHmiAxis => "Simulation".simHmiLinearAxis[12])
   END_RUNG
   RUNG wire#w1
      #"LER_SimAxis+_Axis06_pnp2X"(axisActualPos := "Unit1.Em4.HmiInterface".cmAnodeMainPnP2AxisX.monitoring.actualPosition, pixel := 640, startposition := 0.0, endposition := "Unit1.Em4.HmiInterface".cmAnodeMainPnP2AxisX.configuration.setPositions[0].position, Maxipixel := 120, Minpixel := 0, simHmiAxis => "Simulation".simHmiLinearAxis[6])
      #"LER_SimAxis+_Axis14_pnp2Z"(axisActualPos := "Unit1.Em4.HmiInterface".cmAnodeMainPnP2AxisZ.monitoring.actualPosition, pixel := 234, startposition := 0.0, endposition := "Unit1.Em4.HmiInterface".cmAnodeMainPnP2AxisZ.configuration.setPositions[2].position, Maxipixel := 100, Minpixel :=, simHmiAxis => "Simulation".simHmiLinearAxis[14])
   END_RUNG
   RUNG wire#powerrail
      Contact( #TRUE )
      wire#w2
      #"LER_SimAxis+_Axis07_pnp1X"(axisActualPos := "Unit1.Em5.HmiInterface".cmCathodeMainPnP1AxisX.monitoring.actualPosition, pixel := 400, startposition :=, endposition := "Unit1.Em5.HmiInterface".cmCathodeMainPnP1AxisX.configuration.setPositions[2].position, Maxipixel := 120, Minpixel := 0, simHmiAxis => "Simulation".simHmiLinearAxis[7])
      #"LER_SimAxis+_Axis10_pnp1Z"(axisActualPos := "Unit1.Em5.HmiInterface".cmCathodeMainPnP1AxisZ.monitoring.actualPosition, pixel := 234, startposition :=, endposition := "Unit1.Em5.HmiInterface".cmCathodeMainPnP1AxisZ.configuration.setPositions[2].position, Maxipixel := 100, Minpixel :=, simHmiAxis => "Simulation".simHmiLinearAxis[10])
   END_RUNG
   RUNG wire#w2
      #"LER_SimAxis+_Axis8_pnp2X"(axisActualPos := "Unit1.Em5.HmiInterface".cmCathodeMainPnP2AxisX.monitoring.actualPosition, pixel := 520, startposition := 0.0, endposition := "Unit1.Em5.HmiInterface".cmCathodeMainPnP2AxisX.configuration.setPositions[2].position, Maxipixel := 120, Minpixel := 0, simHmiAxis => "Simulation".simHmiLinearAxis[8])
      #"LER_SimAxis+_Axis13_pnp2Z"(axisActualPos := "Unit1.Em5.HmiInterface".cmCathodeMainPnP2AxisZ.monitoring.actualPosition, pixel := 234, startposition := 0.0, endposition := "Unit1.Em5.HmiInterface".cmCathodeMainPnP2AxisZ.configuration.setPositions[2].position, Maxipixel := 100, Minpixel :=, simHmiAxis => "Simulation".simHmiLinearAxis[13])
   END_RUNG
   RUNG wire#powerrail
      Contact( #TRUE )
      #"LER_SimAxis+_Axis34_cutterX"(axisActualPos := "Unit1.Em7.HmiInterface".cmSepaClampnCutterAxisX.monitoring.actualPosition, pixel := 718, startposition := 0.0, endposition := "Unit1.Em7.HmiInterface".cmSepaClampnCutterAxisX.configuration.setPositions[6].position, Maxipixel := 200, Minpixel :=, simHmiAxis => "Simulation".simHmiLinearAxis[34])
      #"LER_SimAxis+_Axis35_cutterZ"(axisActualPos := "Unit1.Em7.HmiInterface".cmSepaClampnCutterAxisZ.monitoring.actualPosition, pixel := 46, startposition := "Unit1.Em7.HmiInterface".cmSepaClampnCutterAxisZ.configuration.setPositions[3].position, endposition := "Unit1.Em7.HmiInterface".cmSepaClampnCutterAxisZ.configuration.setPositions[1].position, Maxipixel := 55, Minpixel :=, simHmiAxis => "Simulation".simHmiLinearAxis[35])
      #"LER_SimAxis-_Axis36_GripperX"(axisActualPos := "Unit1.Em7.HmiInterface".cmSepaGripperAxisX.monitoring.actualPosition, pixel := 1078, startposition :=, endposition := "Unit1.Em7.HmiInterface".cmSepaGripperAxisX.configuration.setPositions[1].position, Maxipixel := 250, Minpixel :=, simHmiAxis => "Simulation".simHmiLinearAxis[36])
      #"LER_SimAxis+_Axis37_gripperZ"(axisActualPos := "Unit1.Em7.HmiInterface".cmSepaGripperAxisZ.monitoring.actualPosition, pixel := 28, startposition :=, endposition := "Unit1.Em7.HmiInterface".cmSepaGripperAxisZ.configuration.setPositions[1].position, Maxipixel := 55, Minpixel :=, simHmiAxis => "Simulation".simHmiLinearAxis[37])
   END_RUNG
   RUNG wire#powerrail
      Contact( #TRUE )
      #"LER_SimAxis-_Axis32_StackTableZ"(axisActualPos := "Unit1.Em6.HmiInterface".cmStackTableOutFrontAxisZ.monitoring.actualPosition, pixel := 312, startposition :=, endposition := "Unit1.Em6.HmiInterface".cmStackTableOutFrontAxisZ.configuration.setPositions[1].position, Maxipixel := 50, Minpixel :=, simHmiAxis => "Simulation".simHmiLinearAxis[32])
      #"LER_SimAxis+_Axis21_roller"(axisActualPos := "Unit1.Em6.HmiInterface".cmFinalRollerFrontAxisX.monitoring.actualPosition, pixel := 585, startposition :=, endposition := "Unit1.Em7.HmiInterface".cmJRWinderAxisB.configuration.setPositions[3].position, Maxipixel := 115, Minpixel :=, simHmiAxis => "Simulation".simHmiLinearAxis[21])
   END_RUNG
   // the same network as SCL:
   #"LER_SimAxis+_Axis05_pnp1X"(EN := #TRUE,   // "LER_SimAxis+"
                           axisActualPos := "Unit1.Em4.HmiInterface".cmAnodeMainPnP1AxisX.monitoring.actualPosition,
                           pixel := 760,
                           startposition := 0.0,
                           endposition := "Unit1.Em4.HmiInterface".cmAnodeMainPnP1AxisX.configuration.setPositions[0].position,
                           Maxipixel := 120,
                           Minpixel := 0,
                           simHmiAxis => "Simulation".simHmiLinearAxis[5],
                           ENO => #_w1);
   IF #_w1 THEN
       #"LER_SimAxis+_Axis12_pnp1Z"(axisActualPos := "Unit1.Em4.HmiInterface".cmAnodeMainPnP1AxisZ.monitoring.actualPosition,   // "LER_SimAxis+"
                               pixel := 234,
                               endposition := "Unit1.Em4.HmiInterface".cmAnodeMainPnP1AxisZ.configuration.setPositions[2].position,
                               Maxipixel := 100,
                               simHmiAxis => "Simulation".simHmiLinearAxis[12]);
   END_IF;
   #"LER_SimAxis+_Axis06_pnp2X"(EN := #TRUE,   // "LER_SimAxis+"
                           axisActualPos := "Unit1.Em4.HmiInterface".cmAnodeMainPnP2AxisX.monitoring.actualPosition,
                           pixel := 640,
                           startposition := 0.0,
                           endposition := "Unit1.Em4.HmiInterface".cmAnodeMainPnP2AxisX.configuration.setPositions[0].position,
                           Maxipixel := 120,
                           Minpixel := 0,
                           simHmiAxis => "Simulation".simHmiLinearAxis[6],
                           ENO => #_w2);
   IF #_w2 THEN
       #"LER_SimAxis+_Axis14_pnp2Z"(axisActualPos := "Unit1.Em4.HmiInterface".cmAnodeMainPnP2AxisZ.monitoring.actualPosition,   // "LER_SimAxis+"
                               pixel := 234,
                               startposition := 0.0,
                               endposition := "Unit1.Em4.HmiInterface".cmAnodeMainPnP2AxisZ.configuration.setPositions[2].position,
                               Maxipixel := 100,
                               simHmiAxis => "Simulation".simHmiLinearAxis[14]);
   END_IF;
   #"LER_SimAxis+_Axis07_pnp1X"(EN := #TRUE,   // "LER_SimAxis+"
                           axisActualPos := "Unit1.Em5.HmiInterface".cmCathodeMainPnP1AxisX.monitoring.actualPosition,
                           pixel := 400,
                           endposition := "Unit1.Em5.HmiInterface".cmCathodeMainPnP1AxisX.configuration.setPositions[2].position,
                           Maxipixel := 120,
                           Minpixel := 0,
                           simHmiAxis => "Simulation".simHmiLinearAxis[7],
                           ENO => #_w3);
   IF #_w3 THEN
       #"LER_SimAxis+_Axis10_pnp1Z"(axisActualPos := "Unit1.Em5.HmiInterface".cmCathodeMainPnP1AxisZ.monitoring.actualPosition,   // "LER_SimAxis+"
                               pixel := 234,
                               endposition := "Unit1.Em5.HmiInterface".cmCathodeMainPnP1AxisZ.configuration.setPositions[2].position,
                               Maxipixel := 100,
                               simHmiAxis => "Simulation".simHmiLinearAxis[10]);
   END_IF;
   #"LER_SimAxis+_Axis8_pnp2X"(EN := #TRUE,   // "LER_SimAxis+"
                           axisActualPos := "Unit1.Em5.HmiInterface".cmCathodeMainPnP2AxisX.monitoring.actualPosition,
                           pixel := 520,
                           startposition := 0.0,
                           endposition := "Unit1.Em5.HmiInterface".cmCathodeMainPnP2AxisX.configuration.setPositions[2].position,
                           Maxipixel := 120,
                           Minpixel := 0,
                           simHmiAxis => "Simulation".simHmiLinearAxis[8],
                           ENO => #_w4);
   IF #_w4 THEN
       #"LER_SimAxis+_Axis13_pnp2Z"(axisActualPos := "Unit1.Em5.HmiInterface".cmCathodeMainPnP2AxisZ.monitoring.actualPosition,   // "LER_SimAxis+"
                               pixel := 234,
                               startposition := 0.0,
                               endposition := "Unit1.Em5.HmiInterface".cmCathodeMainPnP2AxisZ.configuration.setPositions[2].position,
                               Maxipixel := 100,
                               simHmiAxis => "Simulation".simHmiLinearAxis[13]);
   END_IF;
   #"LER_SimAxis+_Axis34_cutterX"(EN := #TRUE,   // "LER_SimAxis+"
                           axisActualPos := "Unit1.Em7.HmiInterface".cmSepaClampnCutterAxisX.monitoring.actualPosition,
                           pixel := 718,
                           startposition := 0.0,
                           endposition := "Unit1.Em7.HmiInterface".cmSepaClampnCutterAxisX.configuration.setPositions[6].position,
                           Maxipixel := 200,
                           simHmiAxis => "Simulation".simHmiLinearAxis[34],
                           ENO => #_w5);
   #"LER_SimAxis+_Axis35_cutterZ"(EN := #_w5,   // "LER_SimAxis+"
                           axisActualPos := "Unit1.Em7.HmiInterface".cmSepaClampnCutterAxisZ.monitoring.actualPosition,
                           pixel := 46,
                           startposition := "Unit1.Em7.HmiInterface".cmSepaClampnCutterAxisZ.configuration.setPositions[3].position,
                           endposition := "Unit1.Em7.HmiInterface".cmSepaClampnCutterAxisZ.configuration.setPositions[1].position,
                           Maxipixel := 55,
                           simHmiAxis => "Simulation".simHmiLinearAxis[35],
                           ENO => #_w6);
   #"LER_SimAxis-_Axis36_GripperX"(EN := #_w6,   // "LER_SimAxis-"
                           axisActualPos := "Unit1.Em7.HmiInterface".cmSepaGripperAxisX.monitoring.actualPosition,
                           pixel := 1078,
                           endposition := "Unit1.Em7.HmiInterface".cmSepaGripperAxisX.configuration.setPositions[1].position,
                           Maxipixel := 250,
                           simHmiAxis => "Simulation".simHmiLinearAxis[36],
                           ENO => #_w7);
   IF #_w7 THEN
       #"LER_SimAxis+_Axis37_gripperZ"(axisActualPos := "Unit1.Em7.HmiInterface".cmSepaGripperAxisZ.monitoring.actualPosition,   // "LER_SimAxis+"
                               pixel := 28,
                               endposition := "Unit1.Em7.HmiInterface".cmSepaGripperAxisZ.configuration.setPositions[1].position,
                               Maxipixel := 55,
                               simHmiAxis => "Simulation".simHmiLinearAxis[37]);
   END_IF;
   #"LER_SimAxis-_Axis32_StackTableZ"(EN := #TRUE,   // "LER_SimAxis-"
                           axisActualPos := "Unit1.Em6.HmiInterface".cmStackTableOutFrontAxisZ.monitoring.actualPosition,
                           pixel := 312,
                           endposition := "Unit1.Em6.HmiInterface".cmStackTableOutFrontAxisZ.configuration.setPositions[1].position,
                           Maxipixel := 50,
                           simHmiAxis => "Simulation".simHmiLinearAxis[32],
                           ENO => #_w8);
   IF #_w8 THEN
       #"LER_SimAxis+_Axis21_roller"(axisActualPos := "Unit1.Em6.HmiInterface".cmFinalRollerFrontAxisX.monitoring.actualPosition,   // "LER_SimAxis+"
                               pixel := 585,
                               endposition := "Unit1.Em7.HmiInterface".cmJRWinderAxisB.configuration.setPositions[3].position,
                               Maxipixel := 115,
                               simHmiAxis => "Simulation".simHmiLinearAxis[21]);
   END_IF;
END_REGION

REGION Network 4: Simulation Rotary Axis
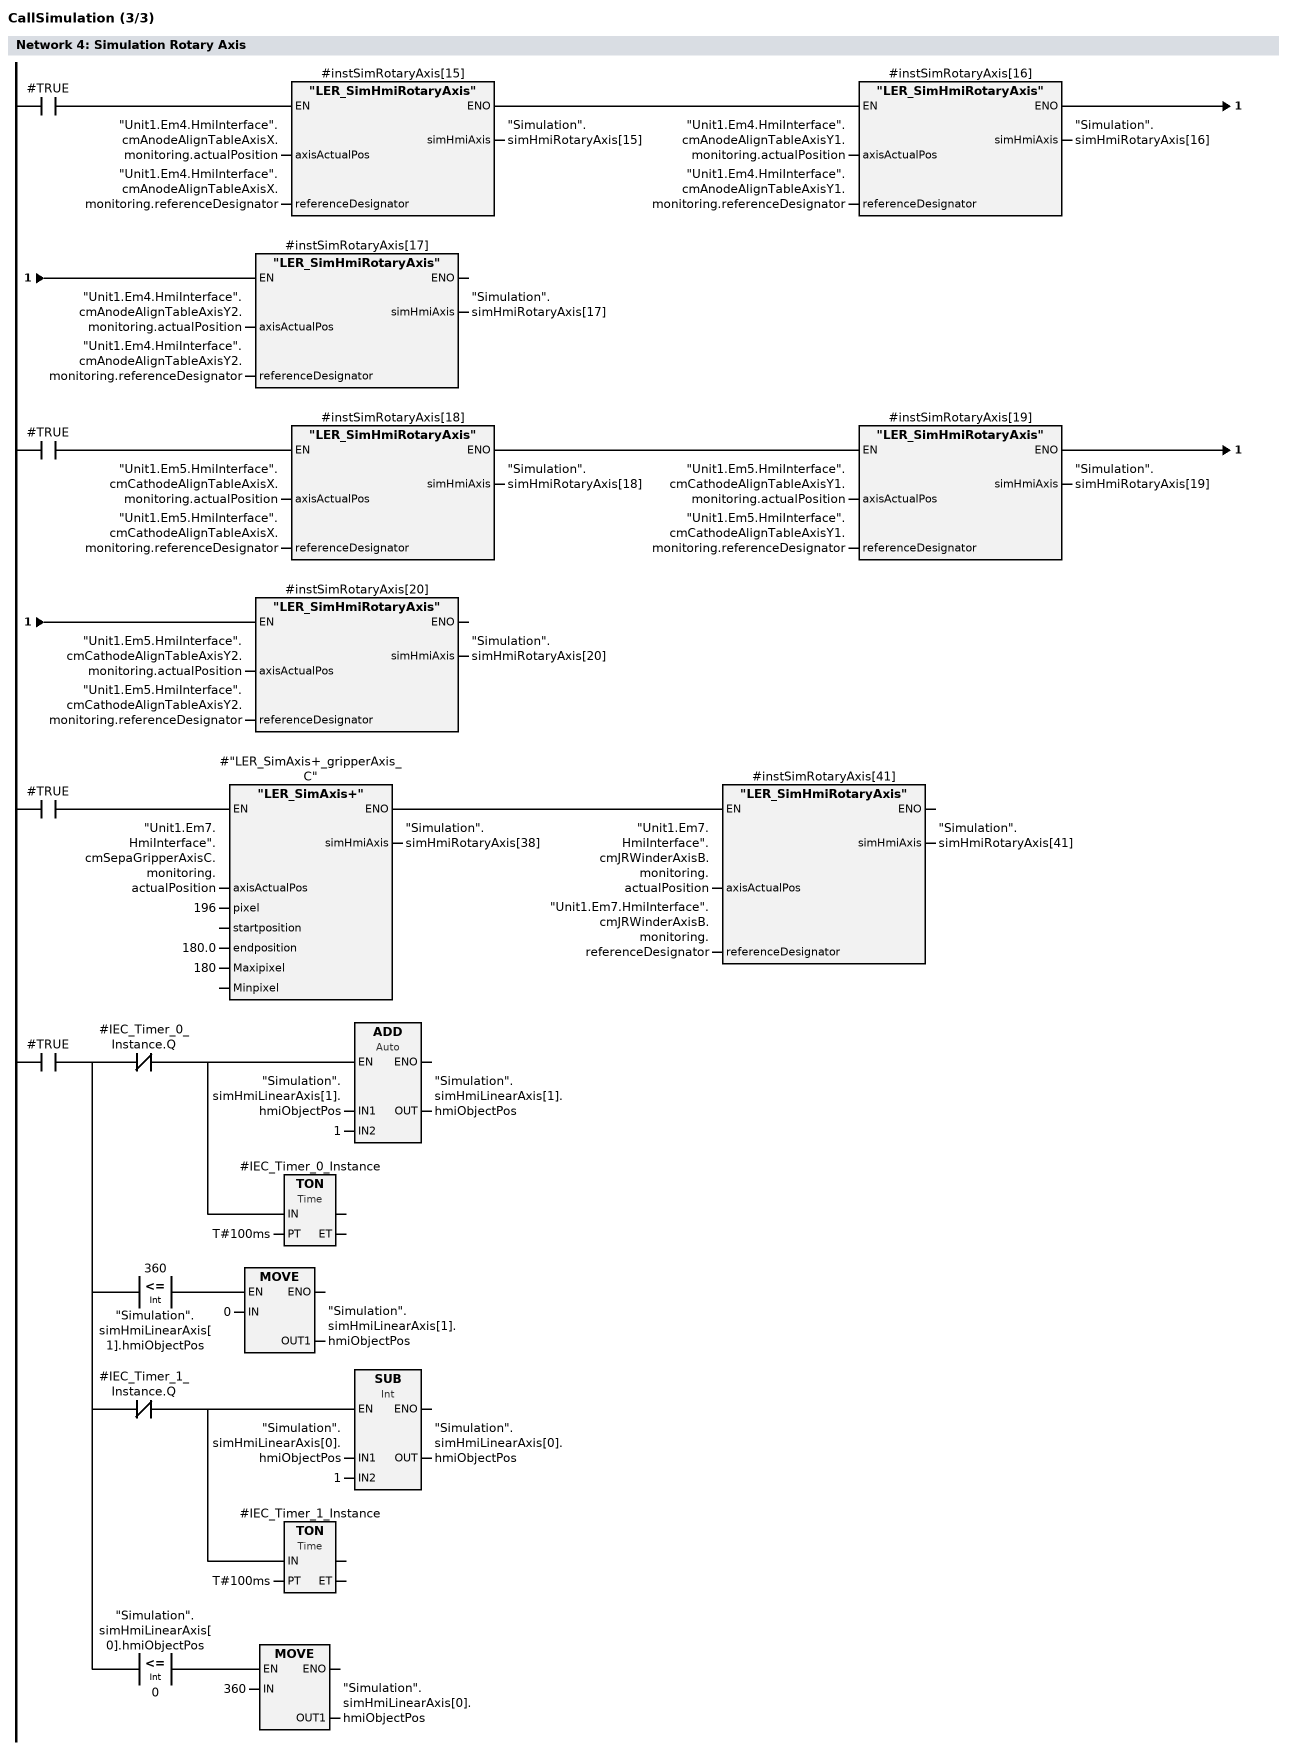
   RUNG wire#powerrail
      Contact( #TRUE )
      #instSimRotaryAxis[15](axisActualPos := "Unit1.Em4.HmiInterface".cmAnodeAlignTableAxisX.monitoring.actualPosition, referenceDesignator := "Unit1.Em4.HmiInterface".cmAnodeAlignTableAxisX.monitoring.referenceDesignator, simHmiAxis => "Simulation".simHmiRotaryAxis[15])
      #instSimRotaryAxis[16](axisActualPos := "Unit1.Em4.HmiInterface".cmAnodeAlignTableAxisY1.monitoring.actualPosition, referenceDesignator := "Unit1.Em4.HmiInterface".cmAnodeAlignTableAxisY1.monitoring.referenceDesignator, simHmiAxis => "Simulation".simHmiRotaryAxis[16])
      #instSimRotaryAxis[17](axisActualPos := "Unit1.Em4.HmiInterface".cmAnodeAlignTableAxisY2.monitoring.actualPosition, referenceDesignator := "Unit1.Em4.HmiInterface".cmAnodeAlignTableAxisY2.monitoring.referenceDesignator, simHmiAxis => "Simulation".simHmiRotaryAxis[17])
   END_RUNG
   RUNG wire#powerrail
      Contact( #TRUE )
      #instSimRotaryAxis[18](axisActualPos := "Unit1.Em5.HmiInterface".cmCathodeAlignTableAxisX.monitoring.actualPosition, referenceDesignator := "Unit1.Em5.HmiInterface".cmCathodeAlignTableAxisX.monitoring.referenceDesignator, simHmiAxis => "Simulation".simHmiRotaryAxis[18])
      #instSimRotaryAxis[19](axisActualPos := "Unit1.Em5.HmiInterface".cmCathodeAlignTableAxisY1.monitoring.actualPosition, referenceDesignator := "Unit1.Em5.HmiInterface".cmCathodeAlignTableAxisY1.monitoring.referenceDesignator, simHmiAxis => "Simulation".simHmiRotaryAxis[19])
      #instSimRotaryAxis[20](axisActualPos := "Unit1.Em5.HmiInterface".cmCathodeAlignTableAxisY2.monitoring.actualPosition, referenceDesignator := "Unit1.Em5.HmiInterface".cmCathodeAlignTableAxisY2.monitoring.referenceDesignator, simHmiAxis => "Simulation".simHmiRotaryAxis[20])
   END_RUNG
   RUNG wire#powerrail
      Contact( #TRUE )
      #"LER_SimAxis+_gripperAxis_C"(axisActualPos := "Unit1.Em7.HmiInterface".cmSepaGripperAxisC.monitoring.actualPosition, pixel := 196, startposition :=, endposition := 180.0, Maxipixel := 180, Minpixel :=, simHmiAxis => "Simulation".simHmiRotaryAxis[38])
      #instSimRotaryAxis[41](axisActualPos := "Unit1.Em7.HmiInterface".cmJRWinderAxisB.monitoring.actualPosition, referenceDesignator := "Unit1.Em7.HmiInterface".cmJRWinderAxisB.monitoring.referenceDesignator, simHmiAxis => "Simulation".simHmiRotaryAxis[41])
   END_RUNG
   RUNG wire#powerrail
      Contact( #TRUE )
      wire#w1
      I_Contact( #IEC_Timer_0_Instance.Q )
      wire#w2
      Add(in1 := "Simulation".simHmiLinearAxis[1].hmiObjectPos, in2 := 1, out => "Simulation".simHmiLinearAxis[1].hmiObjectPos)
   END_RUNG
   RUNG wire#w2
      { S7_Templates := "time_type := Time" } #IEC_Timer_0_Instance.TON(pt := T#100ms, et =>)
   END_RUNG
   RUNG wire#w1
      { S7_Templates := "SrcType := Int" } LE_Contact(in1 := 360, in2 := "Simulation".simHmiLinearAxis[1].hmiObjectPos)
      Move(in := 0, out1 => "Simulation".simHmiLinearAxis[1].hmiObjectPos)
   END_RUNG
   RUNG wire#w1
      I_Contact( #IEC_Timer_1_Instance.Q )
      wire#w3
      { S7_Templates := "SrcType := Int" } Sub(in1 := "Simulation".simHmiLinearAxis[0].hmiObjectPos, in2 := 1, out => "Simulation".simHmiLinearAxis[0].hmiObjectPos)
   END_RUNG
   RUNG wire#w3
      { S7_Templates := "time_type := Time" } #IEC_Timer_1_Instance.TON(pt := T#100ms, et =>)
   END_RUNG
   RUNG wire#w1
      { S7_Templates := "SrcType := Int" } LE_Contact(in1 := "Simulation".simHmiLinearAxis[0].hmiObjectPos, in2 := 0)
      Move(in := 360, out1 => "Simulation".simHmiLinearAxis[0].hmiObjectPos)
   END_RUNG
   // the same network as SCL:
   #instSimRotaryAxis[15](EN := #TRUE,   // "LER_SimHmiRotaryAxis"
                          axisActualPos := "Unit1.Em4.HmiInterface".cmAnodeAlignTableAxisX.monitoring.actualPosition,
                          referenceDesignator := "Unit1.Em4.HmiInterface".cmAnodeAlignTableAxisX.monitoring.referenceDesignator,
                          simHmiAxis => "Simulation".simHmiRotaryAxis[15],
                          ENO => #_w1);
   #instSimRotaryAxis[16](EN := #_w1,   // "LER_SimHmiRotaryAxis"
                          axisActualPos := "Unit1.Em4.HmiInterface".cmAnodeAlignTableAxisY1.monitoring.actualPosition,
                          referenceDesignator := "Unit1.Em4.HmiInterface".cmAnodeAlignTableAxisY1.monitoring.referenceDesignator,
                          simHmiAxis => "Simulation".simHmiRotaryAxis[16],
                          ENO => #_w2);
   IF #_w2 THEN
       #instSimRotaryAxis[17](axisActualPos := "Unit1.Em4.HmiInterface".cmAnodeAlignTableAxisY2.monitoring.actualPosition,   // "LER_SimHmiRotaryAxis"
                              referenceDesignator := "Unit1.Em4.HmiInterface".cmAnodeAlignTableAxisY2.monitoring.referenceDesignator,
                              simHmiAxis => "Simulation".simHmiRotaryAxis[17]);
   END_IF;
   #instSimRotaryAxis[18](EN := #TRUE,   // "LER_SimHmiRotaryAxis"
                          axisActualPos := "Unit1.Em5.HmiInterface".cmCathodeAlignTableAxisX.monitoring.actualPosition,
                          referenceDesignator := "Unit1.Em5.HmiInterface".cmCathodeAlignTableAxisX.monitoring.referenceDesignator,
                          simHmiAxis => "Simulation".simHmiRotaryAxis[18],
                          ENO => #_w3);
   #instSimRotaryAxis[19](EN := #_w3,   // "LER_SimHmiRotaryAxis"
                          axisActualPos := "Unit1.Em5.HmiInterface".cmCathodeAlignTableAxisY1.monitoring.actualPosition,
                          referenceDesignator := "Unit1.Em5.HmiInterface".cmCathodeAlignTableAxisY1.monitoring.referenceDesignator,
                          simHmiAxis => "Simulation".simHmiRotaryAxis[19],
                          ENO => #_w4);
   IF #_w4 THEN
       #instSimRotaryAxis[20](axisActualPos := "Unit1.Em5.HmiInterface".cmCathodeAlignTableAxisY2.monitoring.actualPosition,   // "LER_SimHmiRotaryAxis"
                              referenceDesignator := "Unit1.Em5.HmiInterface".cmCathodeAlignTableAxisY2.monitoring.referenceDesignator,
                              simHmiAxis => "Simulation".simHmiRotaryAxis[20]);
   END_IF;
   #"LER_SimAxis+_gripperAxis_C"(EN := #TRUE,   // "LER_SimAxis+"
                           axisActualPos := "Unit1.Em7.HmiInterface".cmSepaGripperAxisC.monitoring.actualPosition,
                           pixel := 196,
                           endposition := 180.0,
                           Maxipixel := 180,
                           simHmiAxis => "Simulation".simHmiRotaryAxis[38],
                           ENO => #_w5);
   IF #_w5 THEN
       #instSimRotaryAxis[41](axisActualPos := "Unit1.Em7.HmiInterface".cmJRWinderAxisB.monitoring.actualPosition,   // "LER_SimHmiRotaryAxis"
                              referenceDesignator := "Unit1.Em7.HmiInterface".cmJRWinderAxisB.monitoring.referenceDesignator,
                              simHmiAxis => "Simulation".simHmiRotaryAxis[41]);
   END_IF;
   #_w6 := #TRUE AND NOT #IEC_Timer_0_Instance.Q;
   IF #_w6 THEN
       "Simulation".simHmiLinearAxis[1].hmiObjectPos := "Simulation".simHmiLinearAxis[1].hmiObjectPos + 1;
   END_IF;
   #IEC_Timer_0_Instance(IN := #_w6, PT := T#100ms);   // TON
   IF #TRUE AND (360 <= "Simulation".simHmiLinearAxis[1].hmiObjectPos) THEN
       "Simulation".simHmiLinearAxis[1].hmiObjectPos := 0;
   END_IF;
   #_w7 := #TRUE AND NOT #IEC_Timer_1_Instance.Q;
   IF #_w7 THEN
       "Simulation".simHmiLinearAxis[0].hmiObjectPos := "Simulation".simHmiLinearAxis[0].hmiObjectPos - 1;
   END_IF;
   #IEC_Timer_1_Instance(IN := #_w7, PT := T#100ms);   // TON
   IF #TRUE AND ("Simulation".simHmiLinearAxis[0].hmiObjectPos <= 0) THEN
       "Simulation".simHmiLinearAxis[0].hmiObjectPos := 360;
   END_IF;
END_REGION
END_FUNCTION_BLOCK

FUNCTION "CallProductionData" : Void   // FC151, LAD
TITLE = Produktions Daten / Production data
AUTHOR : SICAR
FAMILY : ProdData
VERSION : 1.0
// Dieser Baustein dient als Aufrufschnittstelle für die Funktionsbausteine  
// * _Shiftmodel  
// * _ProdDataCycleTimer  
// * _ProdDataCounter  
// * _ProdDataLimitValues  
// * _ProdDataShiftCounter  
// oder  
// * _ProdDataShiftCounterOee, ShiftProductionTimes
// Call of  FC ProductDataSimulation and LSicar Production Blocks
// stored: IsIECCheckEnabled true, SetENOAutomatically true
   // Ret_Val : Ret_Val
   VAR_TEMP   // added for the SCL form of the ladder/FBD networks
      _w1 : Bool;
      _w2 : Bool;
      _w3 : Bool;
      _w4 : Bool;
      _w5 : Bool;
      _w6 : Bool;
   END_VAR
BEGIN

REGION Network 1: BLOCK INFO HEADER
   // SIEMENS AG / (c)Copyright 2023
   // ------------------------------------------------------------------------------
   // Title:            CallProductionData(FC151)
   // Comment/Function: Call of  FC ProductDataSimulation and LSicar Production Blocks
   // Library/Family:   Automation Framework
   // Author:           Siemens Digital Industry
   // Tested with:      ---
   // Engineering:      TIA Portal V19
   // Restrictions:     -
   // Requirements:     ---
   // ------------------------------------------------------------------------------
   // Change log table:
   // Version  | Date       | Expert in charge       | Changes applied
   // ---------|------------|------------------------|------------------------------
   // 01.00.00 | 11.12.2023 | Siemens Industry Online Support
   //                         First released version
END_REGION

REGION Network 2: Beschreibung / DESCRIPTION
   // **Aufrufschnittstelle**  
   // Der Baustein wird einmalig im zyklischen Programm aufgerufen.  
   // 
   // 
   // #### Weitere Hinweise
   // 
   // #### Updateinfo
   // 
   // #### Weitere Dokumente
   // 
   // ![Icon](_Icon/reference.PNG)
   // 
   // Siehe:  
   // ..\Library Types\LSicar_Shiftmodel.pdf  
   // ..\Library Types\LSicar_ProdDataCycleTimer.pdf  
   // ..\Library Types\LSicar_ProdDataCounter.pdf  
   // ..\Library Types\LSicar_ProdDataLimitValues.pdf  
   // ..\Library Types\LSicar_ProdDataShiftCounter.pdf  
   // ..\Library Types\LSicar_ProdDataShiftCounterOee.pdf  
   // ..\Library Types\LSicar_ShiftProductionTimes.pdf
   // The block is used as a calling interface for the function blocks  
   // *   _Shiftmodel
   // *   _ProdDataCycleTimer
   // *   _ProdDataCounter
   // *   _ProdDataLimitValues
   // *   _ProdDataShiftCounter
   // or
   // *   _ProdDataShiftCounterOee, ShiftProductionTimes
   // 
   // **Calling interface**  
   // The block must be called once only in the cyclic program.  
   // 
   // The block is used as a calling interface for the function blocks  
   // *   _Shiftmodel
   // *   _ProdDataCycleTimer
   // *   _ProdDataCounter
   // *   _ProdDataLimitValues
   // *   _ProdDataShiftCounter
   // or
   // *   _ProdDataShiftCounterOee, ShiftProductionTimes
   // 
   // #### Additional information
   // 
   // #### Update info
   // 
   // #### Further documentations
   // 
   // ![Icon](_Icon/reference.PNG) 
   // 
   // See:  
   // ..\Library Types\LSicar_Shiftmodel.pdf  
   // ..\Library Types\LSicar_ProdDataCycleTimer.pdf  
   // ..\Library Types\LSicar_ProdDataCounter.pdf  
   // ..\Library Types\LSicar_ProdDataLimitValues.pdf  
   // ..\Library Types\LSicar_ProdDataShiftCounter.pdf  
   // ..\Library Types\LSicar_ProdDataShiftCounterOee.pdf  
   // ..\Library Types\LSicar_ShiftProductionTimes.pdf
END_REGION

REGION Network 3: Call Production Simulation
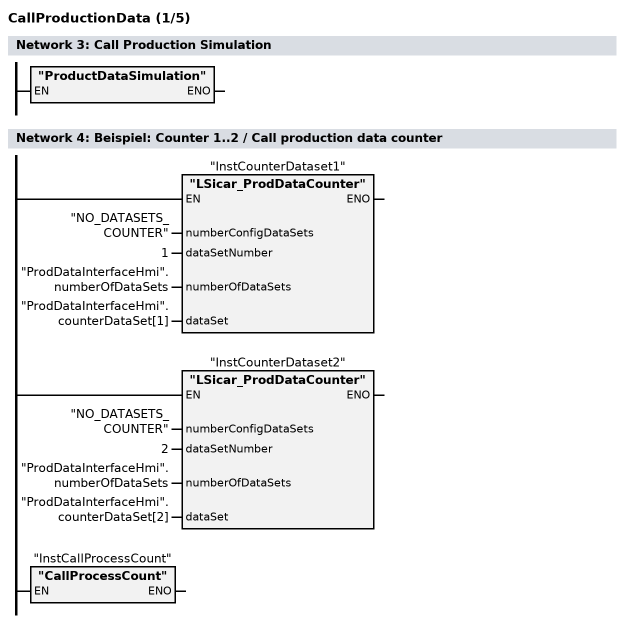
   RUNG wire#powerrail
      "ProductDataSimulation"()
   END_RUNG
   // the same network as SCL:
   "ProductDataSimulation"();
END_REGION

REGION Network 4: Beispiel: Counter 1..2 / Call production data counter
   RUNG wire#powerrail
      "InstCounterDataset1"(numberConfigDataSets := "NO_DATASETS_COUNTER", dataSetNumber := 1, numberOfDataSets := "ProdDataInterfaceHmi".numberOfDataSets, dataSet := "ProdDataInterfaceHmi".counterDataSet[1])
   END_RUNG
   RUNG wire#powerrail
      "InstCounterDataset2"(numberConfigDataSets := "NO_DATASETS_COUNTER", dataSetNumber := 2, numberOfDataSets := "ProdDataInterfaceHmi".numberOfDataSets, dataSet := "ProdDataInterfaceHmi".counterDataSet[2])
   END_RUNG
   RUNG wire#powerrail
      "InstCallProcessCount"()
   END_RUNG
   // the same network as SCL:
   "InstCounterDataset1"(numberConfigDataSets := "NO_DATASETS_COUNTER",   // "LSicar_ProdDataCounter"
                         dataSetNumber := 1,
                         numberOfDataSets := "ProdDataInterfaceHmi".numberOfDataSets,
                         dataSet := "ProdDataInterfaceHmi".counterDataSet[1]);
   "InstCounterDataset2"(numberConfigDataSets := "NO_DATASETS_COUNTER",   // "LSicar_ProdDataCounter"
                         dataSetNumber := 2,
                         numberOfDataSets := "ProdDataInterfaceHmi".numberOfDataSets,
                         dataSet := "ProdDataInterfaceHmi".counterDataSet[2]);
   "InstCallProcessCount"();   // "CallProcessCount"
END_REGION

